LIN {X 0,Y 655.991,Z 1140.634,A -85,B 0,C 180,E1 30861.232,E2 30861.232} C_VEL
LIN {X 0,Y 656.124,Z 1133.603,A -85,B 0,C 180,E1 30859.285,E2 30859.285} C_VEL
LIN {X 0,Y 656.323,Z 1125.528,A -85,B 0,C 180,E1 30857.417,E2 30857.417} C_VEL
LIN {X 0,Y 656.666,Z 1114.351,A -85,B 0,C 180,E1 30855.269,E2 30855.269} C_VEL
LIN {X 0,Y 657.071,Z 1103.391,A -85,B 0,C 180,E1 30853.467,E2 30853.467} C_VEL
LIN {X 0,Y 657.695,Z 1089.324,A -85,B 0,C 180,E1 30851.473,E2 30851.473} C_VEL
LIN {X 0,Y 658.406,Z 1075.305,A -85,B 0,C 180,E1 30849.742,E2 30849.742} C_VEL
LIN {X 0,Y 659.336,Z 1058.307,A -85,B 0,C 180,E1 30847.908,E2 30847.908} C_VEL
LIN {X 0,Y 660.248,Z 1042.797,A -85,B 0,C 180,E1 30846.434,E2 30846.434} C_VEL
LIN {X 0,Y 661.459,Z 1022.865,A -85,B 0,C 180,E1 30844.768,E2 30844.768} C_VEL
LIN {X 0,Y 662.618,Z 1004.407,A -85,B 0,C 180,E1 30843.423,E2 30843.423} C_VEL
LIN {X 0,Y 663.968,Z 982.358,A -85,B 0,C 180,E1 30842.024,E2 30842.024} C_VEL
LIN {X 0,Y 665.114,Z 962.745,A -85,B 0,C 180,E1 30840.949,E2 30840.949} C_VEL
LIN {X 0,Y 666.461,Z 938.728,A -85,B 0,C 180,E1 30839.828,E2 30839.828} C_VEL
LIN {X 0,Y 667.412,Z 919.676,A -85,B 0,C 180,E1 30839.078,E2 30839.078} C_VEL
LIN {X 0,Y 668.429,Z 897.141,A -85,B 0,C 180,E1 30838.328,E2 30838.328} C_VEL
LIN {X 0,Y 669.288,Z 873.179,A -85,B 0,C 180,E1 30837.708,E2 30837.708} C_VEL
LIN {X 0,Y 670.004,Z 850.868,A -85,B 0,C 180,E1 30837.268,E2 30837.268} C_VEL
LIN {X 0,Y 670.501,Z 818.389,A -85,B 0,C 180,E1 30836.831,E2 30836.831} C_VEL
LIN {X 0,Y 672.565,Z 585.869,A -85,B 0,C 180,E1 30834.073,E2 30834.073} C_VEL
LIN {X 0,Y 673.662,Z 473.958,A -85,B 0,C 180,E1 30832.7,E2 30832.7} C_VEL
LIN {X 0,Y 669.198,Z 453.811,A -85,B 0,C 180,E1 30832.148,E2 30832.148} C_VEL
LIN {X 0,Y 669.234,Z 447.014,A -85,B 0,C 180,E1 30831.665,E2 30831.665} C_VEL
LIN {X 0,Y 660.986,Z 426.127,A -85,B 0,C 180,E1 30829.537,E2 30829.537} C_VEL
LIN {X 0,Y 656.734,Z 415.633,A -85,B 0,C 180,E1 30828.38,E2 30828.38} C_VEL
LIN {X 0,Y 656.685,Z 415.429,A -85,B 0,C 180,E1 30825.417,E2 30825.417} C_VEL
LIN {X 0,Y 656.705,Z 415.423,A -85,B 0,C 180,E1 30822.27,E2 30822.27} C_VEL
LIN {X 0,Y 656.674,Z 415.401,A -85,B 0,C 180,E1 30819.304,E2 30819.304} C_VEL
LIN {X 0,Y 656.707,Z 415.43,A -85,B 0,C 180,E1 30816.199,E2 30816.199} C_VEL
LIN {X 0,Y 656.676,Z 415.41,A -85,B 0,C 180,E1 30813.127,E2 30813.127} C_VEL
LIN {X 0,Y 656.705,Z 415.426,A -85,B 0,C 180,E1 30809.961,E2 30809.961} C_VEL
LIN {X 0,Y 656.674,Z 415.427,A -85,B 0,C 180,E1 30806.985,E2 30806.985} C_VEL
LIN {X 0,Y 656.691,Z 415.431,A -85,B 0,C 180,E1 30803.797,E2 30803.797} C_VEL
LIN {X 0,Y 656.667,Z 415.426,A -85,B 0,C 180,E1 30800.874,E2 30800.874} C_VEL
LIN {X 0,Y 656.69,Z 415.425,A -85,B 0,C 180,E1 30797.73,E2 30797.73} C_VEL
LIN {X 0,Y 656.658,Z 415.423,A -85,B 0,C 180,E1 30794.822,E2 30794.822} C_VEL
LIN {X 0,Y 656.692,Z 415.431,A -85,B 0,C 180,E1 30791.684,E2 30791.684} C_VEL
LIN {X 0,Y 656.651,Z 415.427,A -85,B 0,C 180,E1 30788.794,E2 30788.794} C_VEL
LIN {X 0,Y 656.706,Z 415.422,A -85,B 0,C 180,E1 30785.767,E2 30785.767} C_VEL
LIN {X 0,Y 656.64,Z 415.431,A -85,B 0,C 180,E1 30782.88,E2 30782.88} C_VEL
LIN {X 0,Y 656.715,Z 415.418,A -85,B 0,C 180,E1 30779.913,E2 30779.913} C_VEL
LIN {X 0,Y 656.637,Z 415.424,A -85,B 0,C 180,E1 30776.945,E2 30776.945} C_VEL
LIN {X 0,Y 656.657,Z 415.429,A -85,B 0,C 180,E1 30774.232,E2 30774.232} C_VEL
LIN {X 0,Y 656.644,Z 415.432,A -85,B 0,C 180,E1 30771.065,E2 30771.065} C_VEL
LIN {X 0,Y 656.632,Z 415.429,A -85,B 0,C 180,E1 30768.404,E2 30768.404} C_VEL
LIN {X 0,Y 656.685,Z 415.434,A -85,B 0,C 180,E1 30765.359,E2 30765.359} C_VEL
LIN {X 0,Y 656.619,Z 415.429,A -85,B 0,C 180,E1 30762.543,E2 30762.543} C_VEL
LIN {X 0,Y 656.677,Z 415.429,A -85,B 0,C 180,E1 30759.711,E2 30759.711} C_VEL
LIN {X 0,Y 656.619,Z 415.433,A -85,B 0,C 180,E1 30756.671,E2 30756.671} C_VEL
LIN {X 0,Y 656.619,Z 415.433,A -85,B 0,C 180,E1 30754.085,E2 30754.085} C_VEL
LIN {X 0,Y 656.657,Z 415.435,A -85,B 0,C 180,E1 30751.039,E2 30751.039} C_VEL
LIN {X 0,Y 656.603,Z 415.43,A -85,B 0,C 180,E1 30748.349,E2 30748.349} C_VEL
LIN {X 0,Y 656.63,Z 415.433,A -85,B 0,C 180,E1 30745.707,E2 30745.707} C_VEL
LIN {X 0,Y 656.621,Z 415.429,A -85,B 0,C 180,E1 30742.584,E2 30742.584} C_VEL
LIN {X 0,Y 656.627,Z 415.432,A -85,B 0,C 180,E1 30740.609,E2 30740.609} C_VEL
LIN {X 0,Y 655.592,Z 415.557,A -85,B 0,C 180,E1 30739.937,E2 30739.937} C_VEL
LIN {X 0,Y 649.186,Z 416.345,A -85,B 0,C 180,E1 30738.053,E2 30738.053} C_VEL
LIN {X 0,Y 648.701,Z 416.411,A -85,B 0,C 180,E1 30737.563,E2 30737.563} C_VEL
LIN {X 0,Y 648.688,Z 416.395,A -85,B 0,C 180,E1 30734.411,E2 30734.411} C_VEL
LIN {X 0,Y 648.685,Z 416.41,A -85,B 0,C 180,E1 30731.751,E2 30731.751} C_VEL
LIN {X 0,Y 648.793,Z 416.828,A -85,B 0,C 180,E1 30731.291,E2 30731.291} C_VEL
LIN {X 0,Y 657.127,Z 438.059,A -85,B 0,C 180,E1 30728.894,E2 30728.894} C_VEL
LIN {X 0,Y 661.622,Z 449.959,A -85,B 0,C 180,E1 30727.63,E2 30727.63} C_VEL
LIN {X 0,Y 659.646,Z 489.454,A -85,B 0,C 180,E1 30724.693,E2 30724.693} C_VEL
LIN {X 0,Y 659.389,Z 497.949,A -85,B 0,C 180,E1 30724.101,E2 30724.101} C_VEL
LIN {X 0,Y 664.297,Z 521.472,A -85,B 0,C 180,E1 30723.492,E2 30723.492} C_VEL
LIN {X 0,Y 661.38,Z 776.493,A -85,B 0,C 180,E1 30720.424,E2 30720.424} C_VEL
LIN {X 0,Y 660.462,Z 847.868,A -85,B 0,C 180,E1 30719.543,E2 30719.543} C_VEL
LIN {X 0,Y 659.772,Z 870.792,A -85,B 0,C 180,E1 30719.103,E2 30719.103} C_VEL
LIN {X 0,Y 658.928,Z 893.234,A -85,B 0,C 180,E1 30718.525,E2 30718.525} C_VEL
LIN {X 0,Y 657.886,Z 915.745,A -85,B 0,C 180,E1 30717.764,E2 30717.764} C_VEL
LIN {X 0,Y 656.714,Z 938.163,A -85,B 0,C 180,E1 30716.845,E2 30716.845} C_VEL
LIN {X 0,Y 655.667,Z 957.982,A -85,B 0,C 180,E1 30715.874,E2 30715.874} C_VEL
LIN {X 0,Y 654.496,Z 978.096,A -85,B 0,C 180,E1 30714.716,E2 30714.716} C_VEL
LIN {X 0,Y 653.41,Z 996.456,A -85,B 0,C 180,E1 30713.493,E2 30713.493} C_VEL
LIN {X 0,Y 652.29,Z 1014.965,A -85,B 0,C 180,E1 30712.059,E2 30712.059} C_VEL
LIN {X 0,Y 651.303,Z 1032.191,A -85,B 0,C 180,E1 30710.53,E2 30710.53} C_VEL
LIN {X 0,Y 650.415,Z 1047.757,A -85,B 0,C 180,E1 30708.928,E2 30708.928} C_VEL
LIN {X 0,Y 649.633,Z 1063.216,A -85,B 0,C 180,E1 30707.094,E2 30707.094} C_VEL
LIN {X 0,Y 649.074,Z 1075.943,A -85,B 0,C 180,E1 30705.345,E2 30705.345} C_VEL
LIN {X 0,Y 648.61,Z 1087.596,A -85,B 0,C 180,E1 30703.461,E2 30703.461} C_VEL
LIN {X 0,Y 648.305,Z 1097.6,A -85,B 0,C 180,E1 30701.566,E2 30701.566} C_VEL
LIN {X 0,Y 648.095,Z 1105.866,A -85,B 0,C 180,E1 30699.645,E2 30699.645} C_VEL
LIN {X 0,Y 647.972,Z 1112.927,A -85,B 0,C 180,E1 30697.626,E2 30697.626} C_VEL
LIN {X 0,Y 647.918,Z 1117.861,A -85,B 0,C 180,E1 30695.757,E2 30695.757} C_VEL
LIN {X 0,Y 647.899,Z 1121.718,A -85,B 0,C 180,E1 30693.716,E2 30693.716} C_VEL
LIN {X 0,Y 647.9,Z 1123.791,A -85,B 0,C 180,E1 30691.769,E2 30691.769} C_VEL
LIN {X 0,Y 647.896,Z 1124.426,A -85,B 0,C 180,E1 30689.646,E2 30689.646} C_VEL
LIN {X 0,Y 647.904,Z 1123.522,A -85,B 0,C 180,E1 30687.789,E2 30687.789} C_VEL
LIN {X 0,Y 647.909,Z 1120.86,A -85,B 0,C 180,E1 30685.663,E2 30685.663} C_VEL
LIN {X 0,Y 647.945,Z 1117.036,A -85,B 0,C 180,E1 30683.799,E2 30683.799} C_VEL
LIN {X 0,Y 648.021,Z 1110.906,A -85,B 0,C 180,E1 30681.66,E2 30681.66} C_VEL
LIN {X 0,Y 648.137,Z 1103.956,A -85,B 0,C 180,E1 30679.781,E2 30679.781} C_VEL
LIN {X 0,Y 648.371,Z 1094.872,A -85,B 0,C 180,E1 30677.803,E2 30677.803} C_VEL
LIN {X 0,Y 648.727,Z 1084.488,A -85,B 0,C 180,E1 30675.905,E2 30675.905} C_VEL
LIN {X 0,Y 649.19,Z 1072.616,A -85,B 0,C 180,E1 30674.088,E2 30674.088} C_VEL
LIN {X 0,Y 649.858,Z 1058.761,A -85,B 0,C 180,E1 30672.254,E2 30672.254} C_VEL
LIN {X 0,Y 650.604,Z 1044.342,A -85,B 0,C 180,E1 30670.612,E2 30670.612} C_VEL
LIN {X 0,Y 651.564,Z 1027.154,A -85,B 0,C 180,E1 30668.914,E2 30668.914} C_VEL
LIN {X 0,Y 652.618,Z 1009.902,A -85,B 0,C 180,E1 30667.431,E2 30667.431} C_VEL
LIN {X 0,Y 653.681,Z 991.704,A -85,B 0,C 180,E1 30666.087,E2 30666.087} C_VEL
LIN {X 0,Y 654.878,Z 971.864,A -85,B 0,C 180,E1 30664.812,E2 30664.812} C_VEL
LIN {X 0,Y 655.999,Z 951.829,A -85,B 0,C 180,E1 30663.718,E2 30663.718} C_VEL
LIN {X 0,Y 657.164,Z 929.599,A -85,B 0,C 180,E1 30662.695,E2 30662.695} C_VEL
LIN {X 0,Y 658.36,Z 905.845,A -85,B 0,C 180,E1 30661.789,E2 30661.789} C_VEL
LIN {X 0,Y 659.26,Z 884.849,A -85,B 0,C 180,E1 30661.154,E2 30661.154} C_VEL
LIN {X 0,Y 660.066,Z 862.091,A -85,B 0,C 180,E1 30660.619,E2 30660.619} C_VEL
LIN {X 0,Y 660.588,Z 840.006,A -85,B 0,C 180,E1 30660.256,E2 30660.256} C_VEL
LIN {X 0,Y 663.263,Z 610.425,A -85,B 0,C 180,E1 30657.486,E2 30657.486} C_VEL
LIN {X 0,Y 664.119,Z 519.815,A -85,B 0,C 180,E1 30656.386,E2 30656.386} C_VEL
LIN {X 0,Y 659.292,Z 497.129,A -85,B 0,C 180,E1 30655.773,E2 30655.773} C_VEL
LIN {X 0,Y 661.327,Z 455.954,A -85,B 0,C 180,E1 30652.732,E2 30652.732} C_VEL
LIN {X 0,Y 661.489,Z 449.538,A -85,B 0,C 180,E1 30652.238,E2 30652.238} C_VEL
LIN {X 0,Y 653.831,Z 429.55,A -85,B 0,C 180,E1 30650.08,E2 30650.08} C_VEL
LIN {X 0,Y 648.749,Z 416.581,A -85,B 0,C 180,E1 30648.569,E2 30648.569} C_VEL
LIN {X 0,Y 648.685,Z 416.396,A -85,B 0,C 180,E1 30645.788,E2 30645.788} C_VEL
LIN {X 0,Y 648.762,Z 416.412,A -85,B 0,C 180,E1 30642.808,E2 30642.808} C_VEL
LIN {X 0,Y 648.677,Z 416.419,A -85,B 0,C 180,E1 30639.884,E2 30639.884} C_VEL
LIN {X 0,Y 648.697,Z 416.411,A -85,B 0,C 180,E1 30637.284,E2 30637.284} C_VEL
LIN {X 0,Y 648.689,Z 416.424,A -85,B 0,C 180,E1 30634.13,E2 30634.13} C_VEL
LIN {X 0,Y 648.671,Z 416.419,A -85,B 0,C 180,E1 30631.504,E2 30631.504} C_VEL
LIN {X 0,Y 648.745,Z 416.415,A -85,B 0,C 180,E1 30628.535,E2 30628.535} C_VEL
LIN {X 0,Y 648.664,Z 416.424,A -85,B 0,C 180,E1 30625.61,E2 30625.61} C_VEL
LIN {X 0,Y 648.719,Z 416.423,A -85,B 0,C 180,E1 30622.821,E2 30622.821} C_VEL
LIN {X 0,Y 648.683,Z 416.422,A -85,B 0,C 180,E1 30619.823,E2 30619.823} C_VEL
LIN {X 0,Y 648.679,Z 416.419,A -85,B 0,C 180,E1 30617.215,E2 30617.215} C_VEL
LIN {X 0,Y 648.742,Z 416.418,A -85,B 0,C 180,E1 30614.186,E2 30614.186} C_VEL
LIN {X 0,Y 648.682,Z 416.42,A -85,B 0,C 180,E1 30611.378,E2 30611.378} C_VEL
LIN {X 0,Y 648.746,Z 416.412,A -85,B 0,C 180,E1 30608.509,E2 30608.509} C_VEL
LIN {X 0,Y 648.695,Z 416.42,A -85,B 0,C 180,E1 30605.484,E2 30605.484} C_VEL
LIN {X 0,Y 648.713,Z 416.413,A -85,B 0,C 180,E1 30602.739,E2 30602.739} C_VEL
LIN {X 0,Y 648.711,Z 416.409,A -85,B 0,C 180,E1 30599.558,E2 30599.558} C_VEL
LIN {X 0,Y 648.707,Z 416.422,A -85,B 0,C 180,E1 30596.819,E2 30596.819} C_VEL
LIN {X 0,Y 648.749,Z 416.415,A -85,B 0,C 180,E1 30593.718,E2 30593.718} C_VEL
LIN {X 0,Y 648.707,Z 416.418,A -85,B 0,C 180,E1 30590.865,E2 30590.865} C_VEL
LIN {X 0,Y 648.772,Z 416.415,A -85,B 0,C 180,E1 30587.81,E2 30587.81} C_VEL
LIN {X 0,Y 648.711,Z 416.414,A -85,B 0,C 180,E1 30584.901,E2 30584.901} C_VEL
LIN {X 0,Y 648.77,Z 416.408,A -85,B 0,C 180,E1 30581.954,E2 30581.954} C_VEL
LIN {X 0,Y 648.721,Z 416.416,A -85,B 0,C 180,E1 30578.953,E2 30578.953} C_VEL
LIN {X 0,Y 648.77,Z 416.421,A -85,B 0,C 180,E1 30575.991,E2 30575.991} C_VEL
LIN {X 0,Y 648.727,Z 416.417,A -85,B 0,C 180,E1 30572.856,E2 30572.856} C_VEL
LIN {X 0,Y 648.773,Z 416.414,A -85,B 0,C 180,E1 30569.941,E2 30569.941} C_VEL
LIN {X 0,Y 648.733,Z 416.396,A -85,B 0,C 180,E1 30566.817,E2 30566.817} C_VEL
LIN {X 0,Y 648.766,Z 416.418,A -85,B 0,C 180,E1 30563.822,E2 30563.822} C_VEL
LIN {X 0,Y 648.732,Z 416.388,A -85,B 0,C 180,E1 30560.691,E2 30560.691} C_VEL
LIN {X 0,Y 648.765,Z 416.41,A -85,B 0,C 180,E1 30557.661,E2 30557.661} C_VEL
LIN {X 0,Y 648.744,Z 416.419,A -85,B 0,C 180,E1 30554.53,E2 30554.53} C_VEL
LIN {X 0,Y 648.775,Z 416.622,A -85,B 0,C 180,E1 30552.156,E2 30552.156} C_VEL
LIN {X 0,Y 657.494,Z 438.049,A -85,B 0,C 180,E1 30549.81,E2 30549.81} C_VEL
LIN {X 0,Y 662.5,Z 451.205,A -85,B 0,C 180,E1 30548.477,E2 30548.477} C_VEL
LIN {X 0,Y 662.507,Z 454.848,A -85,B 0,C 180,E1 30548.253,E2 30548.253} C_VEL
LIN {X 0,Y 667.304,Z 477.152,A -85,B 0,C 180,E1 30547.654,E2 30547.654} C_VEL
LIN {X 0,Y 664.523,Z 721.617,A -85,B 0,C 180,E1 30544.669,E2 30544.669} C_VEL
LIN {X 0,Y 663.232,Z 844.483,A -85,B 0,C 180,E1 30543.181,E2 30543.181} C_VEL
LIN {X 0,Y 662.513,Z 870.087,A -85,B 0,C 180,E1 30542.714,E2 30542.714} C_VEL
LIN {X 0,Y 661.751,Z 891.398,A -85,B 0,C 180,E1 30542.194,E2 30542.194} C_VEL
LIN {X 0,Y 660.735,Z 914.535,A -85,B 0,C 180,E1 30541.473,E2 30541.473} C_VEL
LIN {X 0,Y 659.605,Z 935.33,A -85,B 0,C 180,E1 30540.671,E2 30540.671} C_VEL
LIN {X 0,Y 658.38,Z 957.268,A -85,B 0,C 180,E1 30539.677,E2 30539.677} C_VEL
LIN {X 0,Y 656.936,Z 979.114,A -85,B 0,C 180,E1 30538.5,E2 30538.5} C_VEL
LIN {X 0,Y 655.616,Z 999.646,A -85,B 0,C 180,E1 30537.228,E2 30537.228} C_VEL
LIN {X 0,Y 654.268,Z 1019.215,A -85,B 0,C 180,E1 30535.821,E2 30535.821} C_VEL
LIN {X 0,Y 653.067,Z 1037.201,A -85,B 0,C 180,E1 30534.357,E2 30534.357} C_VEL
LIN {X 0,Y 651.924,Z 1054.602,A -85,B 0,C 180,E1 30532.737,E2 30532.737} C_VEL
LIN {X 0,Y 650.985,Z 1069.628,A -85,B 0,C 180,E1 30531.159,E2 30531.159} C_VEL
LIN {X 0,Y 650.057,Z 1086.032,A -85,B 0,C 180,E1 30529.19,E2 30529.19} C_VEL
LIN {X 0,Y 649.404,Z 1099.154,A -85,B 0,C 180,E1 30527.38,E2 30527.38} C_VEL
LIN {X 0,Y 648.819,Z 1112.382,A -85,B 0,C 180,E1 30525.263,E2 30525.263} C_VEL
LIN {X 0,Y 648.448,Z 1122.48,A -85,B 0,C 180,E1 30523.373,E2 30523.373} C_VEL
LIN {X 0,Y 648.165,Z 1132.189,A -85,B 0,C 180,E1 30521.208,E2 30521.208} C_VEL
LIN {X 0,Y 648.053,Z 1138.817,A -85,B 0,C 180,E1 30519.413,E2 30519.413} C_VEL
LIN {X 0,Y 647.946,Z 1145.243,A -85,B 0,C 180,E1 30517.27,E2 30517.27} C_VEL
LIN {X 0,Y 647.896,Z 1149.656,A -85,B 0,C 180,E1 30515.224,E2 30515.224} C_VEL
LIN {X 0,Y 647.904,Z 1152.463,A -85,B 0,C 180,E1 30513.362,E2 30513.362} C_VEL
LIN {X 0,Y 647.909,Z 1154.215,A -85,B 0,C 180,E1 30511.15,E2 30511.15} C_VEL
LIN {X 0,Y 647.885,Z 1154.328,A -85,B 0,C 180,E1 30509.293,E2 30509.293} C_VEL
LIN {X 0,Y 647.888,Z 1153.225,A -85,B 0,C 180,E1 30507.346,E2 30507.346} C_VEL
LIN {X 0,Y 647.903,Z 1150.292,A -85,B 0,C 180,E1 30505.131,E2 30505.131} C_VEL
LIN {X 0,Y 647.939,Z 1146.689,A -85,B 0,C 180,E1 30503.354,E2 30503.354} C_VEL
LIN {X 0,Y 648,Z 1140.935,A -85,B 0,C 180,E1 30501.213,E2 30501.213} C_VEL
LIN {X 0,Y 648.142,Z 1133.603,A -85,B 0,C 180,E1 30499.152,E2 30499.152} C_VEL
LIN {X 0,Y 648.372,Z 1125.529,A -85,B 0,C 180,E1 30497.26,E2 30497.26} C_VEL
LIN {X 0,Y 648.748,Z 1114.436,A -85,B 0,C 180,E1 30495.1,E2 30495.1} C_VEL
LIN {X 0,Y 649.198,Z 1103.393,A -85,B 0,C 180,E1 30493.261,E2 30493.261} C_VEL
LIN {X 0,Y 649.877,Z 1089.323,A -85,B 0,C 180,E1 30491.242,E2 30491.242} C_VEL
LIN {X 0,Y 650.67,Z 1075.307,A -85,B 0,C 180,E1 30489.49,E2 30489.49} C_VEL
LIN {X 0,Y 651.686,Z 1058.305,A -85,B 0,C 180,E1 30487.635,E2 30487.635} C_VEL
LIN {X 0,Y 652.726,Z 1042.29,A -85,B 0,C 180,E1 30486.098,E2 30486.098} C_VEL
LIN {X 0,Y 654.04,Z 1022.359,A -85,B 0,C 180,E1 30484.421,E2 30484.421} C_VEL
LIN {X 0,Y 655.275,Z 1004.392,A -85,B 0,C 180,E1 30483.1,E2 30483.1} C_VEL
LIN {X 0,Y 656.73,Z 982.354,A -85,B 0,C 180,E1 30481.688,E2 30481.688} C_VEL
LIN {X 0,Y 657.988,Z 962.741,A -85,B 0,C 180,E1 30480.604,E2 30480.604} C_VEL
LIN {X 0,Y 659.437,Z 938.724,A -85,B 0,C 180,E1 30479.472,E2 30479.472} C_VEL
LIN {X 0,Y 660.468,Z 919.672,A -85,B 0,C 180,E1 30478.716,E2 30478.716} C_VEL
LIN {X 0,Y 661.503,Z 898.098,A -85,B 0,C 180,E1 30477.993,E2 30477.993} C_VEL
LIN {X 0,Y 662.367,Z 873.835,A -85,B 0,C 180,E1 30477.367,E2 30477.367} C_VEL
LIN {X 0,Y 663.055,Z 851.771,A -85,B 0,C 180,E1 30476.935,E2 30476.935} C_VEL
LIN {X 0,Y 663.553,Z 819.351,A -85,B 0,C 180,E1 30476.498,E2 30476.498} C_VEL
LIN {X 0,Y 665.842,Z 590.197,A -85,B 0,C 180,E1 30473.746,E2 30473.746} C_VEL
LIN {X 0,Y 667.088,Z 475.51,A -85,B 0,C 180,E1 30472.318,E2 30472.318} C_VEL
LIN {X 0,Y 662.402,Z 454.038,A -85,B 0,C 180,E1 30471.715,E2 30471.715} C_VEL
LIN {X 0,Y 662.299,Z 450.377,A -85,B 0,C 180,E1 30471.448,E2 30471.448} C_VEL
LIN {X 0,Y 654.091,Z 429.742,A -85,B 0,C 180,E1 30469.308,E2 30469.308} C_VEL
LIN {X 0,Y 648.773,Z 416.612,A -85,B 0,C 180,E1 30467.839,E2 30467.839} C_VEL
LIN {X 0,Y 648.763,Z 416.396,A -85,B 0,C 180,E1 30464.777,E2 30464.777} C_VEL
LIN {X 0,Y 648.743,Z 416.422,A -85,B 0,C 180,E1 30461.746,E2 30461.746} C_VEL
LIN {X 0,Y 648.767,Z 416.388,A -85,B 0,C 180,E1 30458.736,E2 30458.736} C_VEL
LIN {X 0,Y 648.736,Z 416.411,A -85,B 0,C 180,E1 30455.634,E2 30455.634} C_VEL
LIN {X 0,Y 648.767,Z 416.398,A -85,B 0,C 180,E1 30452.54,E2 30452.54} C_VEL
LIN {X 0,Y 648.733,Z 416.412,A -85,B 0,C 180,E1 30449.552,E2 30449.552} C_VEL
LIN {X 0,Y 648.768,Z 416.414,A -85,B 0,C 180,E1 30446.548,E2 30446.548} C_VEL
LIN {X 0,Y 648.725,Z 416.417,A -85,B 0,C 180,E1 30443.432,E2 30443.432} C_VEL
LIN {X 0,Y 648.767,Z 416.413,A -85,B 0,C 180,E1 30440.436,E2 30440.436} C_VEL
LIN {X 0,Y 648.721,Z 416.419,A -85,B 0,C 180,E1 30437.306,E2 30437.306} C_VEL
LIN {X 0,Y 648.763,Z 416.409,A -85,B 0,C 180,E1 30434.367,E2 30434.367} C_VEL
LIN {X 0,Y 648.718,Z 416.417,A -85,B 0,C 180,E1 30431.289,E2 30431.289} C_VEL
LIN {X 0,Y 648.738,Z 416.414,A -85,B 0,C 180,E1 30428.42,E2 30428.42} C_VEL
LIN {X 0,Y 648.719,Z 416.414,A -85,B 0,C 180,E1 30425.306,E2 30425.306} C_VEL
LIN {X 0,Y 648.719,Z 416.418,A -85,B 0,C 180,E1 30422.474,E2 30422.474} C_VEL
LIN {X 0,Y 648.714,Z 416.422,A -85,B 0,C 180,E1 30419.205,E2 30419.205} C_VEL
LIN {X 0,Y 648.704,Z 416.41,A -85,B 0,C 180,E1 30416.465,E2 30416.465} C_VEL
LIN {X 0,Y 648.735,Z 416.418,A -85,B 0,C 180,E1 30413.362,E2 30413.362} C_VEL
LIN {X 0,Y 648.69,Z 416.419,A -85,B 0,C 180,E1 30410.575,E2 30410.575} C_VEL
LIN {X 0,Y 648.768,Z 416.41,A -85,B 0,C 180,E1 30407.63,E2 30407.63} C_VEL
LIN {X 0,Y 648.685,Z 416.422,A -85,B 0,C 180,E1 30404.717,E2 30404.717} C_VEL
LIN {X 0,Y 648.703,Z 416.417,A -85,B 0,C 180,E1 30402.045,E2 30402.045} C_VEL
LIN {X 0,Y 648.69,Z 416.42,A -85,B 0,C 180,E1 30398.836,E2 30398.836} C_VEL
LIN {X 0,Y 648.676,Z 416.422,A -85,B 0,C 180,E1 30396.277,E2 30396.277} C_VEL
LIN {X 0,Y 648.758,Z 416.422,A -85,B 0,C 180,E1 30393.352,E2 30393.352} C_VEL
LIN {X 0,Y 648.668,Z 416.426,A -85,B 0,C 180,E1 30390.444,E2 30390.444} C_VEL
LIN {X 0,Y 648.679,Z 416.419,A -85,B 0,C 180,E1 30387.873,E2 30387.873} C_VEL
LIN {X 0,Y 648.677,Z 416.397,A -85,B 0,C 180,E1 30384.629,E2 30384.629} C_VEL
LIN {X 0,Y 648.671,Z 416.423,A -85,B 0,C 180,E1 30381.969,E2 30381.969} C_VEL
LIN {X 0,Y 648.75,Z 416.39,A -85,B 0,C 180,E1 30379.045,E2 30379.045} C_VEL
LIN {X 0,Y 648.701,Z 416.411,A -85,B 0,C 180,E1 30377.563,E2 30377.563} C_VEL
LIN {X 0,Y 647.769,Z 416.544,A -85,B 0,C 180,E1 30376.882,E2 30376.882} C_VEL
LIN {X 0,Y 641.223,Z 417.33,A -85,B 0,C 180,E1 30374.926,E2 30374.926} C_VEL
LIN {X 0,Y 640.754,Z 417.382,A -85,B 0,C 180,E1 30374.479,E2 30374.479} C_VEL
LIN {X 0,Y 640.771,Z 417.624,A -85,B 0,C 180,E1 30371.884,E2 30371.884} C_VEL
LIN {X 0,Y 647.744,Z 434.924,A -85,B 0,C 180,E1 30369.838,E2 30369.838} C_VEL
LIN {X 0,Y 654.667,Z 453.446,A -85,B 0,C 180,E1 30367.829,E2 30367.829} C_VEL
LIN {X 0,Y 652.477,Z 493.787,A -85,B 0,C 180,E1 30364.804,E2 30364.804} C_VEL
LIN {X 0,Y 652.502,Z 497.976,A -85,B 0,C 180,E1 30364.541,E2 30364.541} C_VEL
LIN {X 0,Y 657.764,Z 522.777,A -85,B 0,C 180,E1 30363.881,E2 30363.881} C_VEL
LIN {X 0,Y 654.701,Z 777.349,A -85,B 0,C 180,E1 30360.801,E2 30360.801} C_VEL
LIN {X 0,Y 653.739,Z 847.737,A -85,B 0,C 180,E1 30359.926,E2 30359.926} C_VEL
LIN {X 0,Y 653.008,Z 870.705,A -85,B 0,C 180,E1 30359.485,E2 30359.485} C_VEL
LIN {X 0,Y 652.101,Z 893.018,A -85,B 0,C 180,E1 30358.908,E2 30358.908} C_VEL
LIN {X 0,Y 651.019,Z 914.402,A -85,B 0,C 180,E1 30358.183,E2 30358.183} C_VEL
LIN {X 0,Y 649.85,Z 935.051,A -85,B 0,C 180,E1 30357.341,E2 30357.341} C_VEL
LIN {X 0,Y 648.508,Z 955.763,A -85,B 0,C 180,E1 30356.313,E2 30356.313} C_VEL
LIN {X 0,Y 647.181,Z 976.91,A -85,B 0,C 180,E1 30355.094,E2 30355.094} C_VEL
LIN {X 0,Y 645.987,Z 995.125,A -85,B 0,C 180,E1 30353.876,E2 30353.876} C_VEL
LIN {X 0,Y 644.782,Z 1013.861,A -85,B 0,C 180,E1 30352.426,E2 30352.426} C_VEL
LIN {X 0,Y 643.707,Z 1030.678,A -85,B 0,C 180,E1 30350.933,E2 30350.933} C_VEL
LIN {X 0,Y 642.762,Z 1046.071,A -85,B 0,C 180,E1 30349.351,E2 30349.351} C_VEL
LIN {X 0,Y 641.976,Z 1060.383,A -85,B 0,C 180,E1 30347.681,E2 30347.681} C_VEL
LIN {X 0,Y 641.29,Z 1073.264,A -85,B 0,C 180,E1 30345.927,E2 30345.927} C_VEL
LIN {X 0,Y 640.763,Z 1085.535,A -85,B 0,C 180,E1 30343.997,E2 30343.997} C_VEL
LIN {X 0,Y 640.407,Z 1095.334,A -85,B 0,C 180,E1 30342.168,E2 30342.168} C_VEL
LIN {X 0,Y 640.141,Z 1104.666,A -85,B 0,C 180,E1 30340.075,E2 30340.075} C_VEL
LIN {X 0,Y 640.017,Z 1111.514,A -85,B 0,C 180,E1 30338.173,E2 30338.173} C_VEL
LIN {X 0,Y 639.943,Z 1117.24,A -85,B 0,C 180,E1 30336.099,E2 30336.099} C_VEL
LIN {X 0,Y 639.913,Z 1121.019,A -85,B 0,C 180,E1 30334.212,E2 30334.212} C_VEL
LIN {X 0,Y 639.906,Z 1123.518,A -85,B 0,C 180,E1 30332.149,E2 30332.149} C_VEL
LIN {X 0,Y 639.903,Z 1124.448,A -85,B 0,C 180,E1 30330.179,E2 30330.179} C_VEL
LIN {X 0,Y 639.903,Z 1123.793,A -85,B 0,C 180,E1 30328.12,E2 30328.12} C_VEL
LIN {X 0,Y 639.905,Z 1121.72,A -85,B 0,C 180,E1 30326.147,E2 30326.147} C_VEL
LIN {X 0,Y 639.928,Z 1117.86,A -85,B 0,C 180,E1 30324.081,E2 30324.081} C_VEL
LIN {X 0,Y 639.986,Z 1112.673,A -85,B 0,C 180,E1 30322.097,E2 30322.097} C_VEL
LIN {X 0,Y 640.116,Z 1105.723,A -85,B 0,C 180,E1 30320.106,E2 30320.106} C_VEL
LIN {X 0,Y 640.344,Z 1097.595,A -85,B 0,C 180,E1 30318.196,E2 30318.196} C_VEL
LIN {X 0,Y 640.681,Z 1087.588,A -85,B 0,C 180,E1 30316.277,E2 30316.277} C_VEL
LIN {X 0,Y 641.17,Z 1076.426,A -85,B 0,C 180,E1 30314.441,E2 30314.441} C_VEL
LIN {X 0,Y 641.773,Z 1063.874,A -85,B 0,C 180,E1 30312.688,E2 30312.688} C_VEL
LIN {X 0,Y 642.572,Z 1049.415,A -85,B 0,C 180,E1 30310.927,E2 30310.927} C_VEL
LIN {X 0,Y 643.478,Z 1034.403,A -85,B 0,C 180,E1 30309.345,E2 30309.345} C_VEL
LIN {X 0,Y 644.603,Z 1016.532,A -85,B 0,C 180,E1 30307.709,E2 30307.709} C_VEL
LIN {X 0,Y 645.807,Z 998.347,A -85,B 0,C 180,E1 30306.262,E2 30306.262} C_VEL
LIN {X 0,Y 646.985,Z 979.741,A -85,B 0,C 180,E1 30304.996,E2 30304.996} C_VEL
LIN {X 0,Y 648.297,Z 959.455,A -85,B 0,C 180,E1 30303.794,E2 30303.794} C_VEL
LIN {X 0,Y 649.514,Z 939.785,A -85,B 0,C 180,E1 30302.792,E2 30302.792} C_VEL
LIN {X 0,Y 650.842,Z 917.92,A -85,B 0,C 180,E1 30301.859,E2 30301.859} C_VEL
LIN {X 0,Y 651.836,Z 898.37,A -85,B 0,C 180,E1 30301.174,E2 30301.174} C_VEL
LIN {X 0,Y 652.833,Z 875.117,A -85,B 0,C 180,E1 30300.526,E2 30300.526} C_VEL
LIN {X 0,Y 653.552,Z 853.926,A -85,B 0,C 180,E1 30300.088,E2 30300.088} C_VEL
LIN {X 0,Y 654.137,Z 823.568,A -85,B 0,C 180,E1 30299.667,E2 30299.667} C_VEL
LIN {X 0,Y 656.911,Z 591.86,A -85,B 0,C 180,E1 30296.864,E2 30296.864} C_VEL
LIN {X 0,Y 657.58,Z 521.351,A -85,B 0,C 180,E1 30295.999,E2 30295.999} C_VEL
LIN {X 0,Y 652.34,Z 496.691,A -85,B 0,C 180,E1 30295.316,E2 30295.316} C_VEL
LIN {X 0,Y 654.5,Z 456.495,A -85,B 0,C 180,E1 30292.313,E2 30292.313} C_VEL
LIN {X 0,Y 654.531,Z 452.855,A -85,B 0,C 180,E1 30292.024,E2 30292.024} C_VEL
LIN {X 0,Y 646.997,Z 433.261,A -85,B 0,C 180,E1 30289.876,E2 30289.876} C_VEL
LIN {X 0,Y 641.853,Z 420.538,A -85,B 0,C 180,E1 30288.396,E2 30288.396} C_VEL
LIN {X 0,Y 640.771,Z 417.564,A -85,B 0,C 180,E1 30288.006,E2 30288.006} C_VEL
LIN {X 0,Y 640.788,Z 417.379,A -85,B 0,C 180,E1 30285.234,E2 30285.234} C_VEL
LIN {X 0,Y 640.747,Z 417.395,A -85,B 0,C 180,E1 30282.146,E2 30282.146} C_VEL
LIN {X 0,Y 640.744,Z 417.408,A -85,B 0,C 180,E1 30279.546,E2 30279.546} C_VEL
LIN {X 0,Y 640.784,Z 417.377,A -85,B 0,C 180,E1 30276.479,E2 30276.479} C_VEL
LIN {X 0,Y 640.733,Z 417.413,A -85,B 0,C 180,E1 30273.642,E2 30273.642} C_VEL
LIN {X 0,Y 640.819,Z 417.404,A -85,B 0,C 180,E1 30270.679,E2 30270.679} C_VEL
LIN {X 0,Y 640.725,Z 417.41,A -85,B 0,C 180,E1 30267.713,E2 30267.713} C_VEL
LIN {X 0,Y 640.769,Z 417.408,A -85,B 0,C 180,E1 30264.918,E2 30264.918} C_VEL
LIN {X 0,Y 640.743,Z 417.409,A -85,B 0,C 180,E1 30261.899,E2 30261.899} C_VEL
LIN {X 0,Y 640.741,Z 417.412,A -85,B 0,C 180,E1 30259.225,E2 30259.225} C_VEL
LIN {X 0,Y 640.787,Z 417.407,A -85,B 0,C 180,E1 30256.126,E2 30256.126} C_VEL
LIN {X 0,Y 640.74,Z 417.408,A -85,B 0,C 180,E1 30253.354,E2 30253.354} C_VEL
LIN {X 0,Y 640.821,Z 417.411,A -85,B 0,C 180,E1 30250.428,E2 30250.428} C_VEL
LIN {X 0,Y 640.75,Z 417.404,A -85,B 0,C 180,E1 30247.442,E2 30247.442} C_VEL
LIN {X 0,Y 640.776,Z 417.411,A -85,B 0,C 180,E1 30244.744,E2 30244.744} C_VEL
LIN {X 0,Y 640.767,Z 417.409,A -85,B 0,C 180,E1 30241.52,E2 30241.52} C_VEL
LIN {X 0,Y 640.765,Z 417.399,A -85,B 0,C 180,E1 30238.838,E2 30238.838} C_VEL
LIN {X 0,Y 640.801,Z 417.4,A -85,B 0,C 180,E1 30235.705,E2 30235.705} C_VEL
LIN {X 0,Y 640.765,Z 417.408,A -85,B 0,C 180,E1 30232.919,E2 30232.919} C_VEL
LIN {X 0,Y 640.829,Z 417.398,A -85,B 0,C 180,E1 30229.845,E2 30229.845} C_VEL
LIN {X 0,Y 640.771,Z 417.407,A -85,B 0,C 180,E1 30226.923,E2 30226.923} C_VEL
LIN {X 0,Y 640.835,Z 417.407,A -85,B 0,C 180,E1 30223.968,E2 30223.968} C_VEL
LIN {X 0,Y 640.777,Z 417.402,A -85,B 0,C 180,E1 30220.871,E2 30220.871} C_VEL
LIN {X 0,Y 640.835,Z 417.397,A -85,B 0,C 180,E1 30217.912,E2 30217.912} C_VEL
LIN {X 0,Y 640.785,Z 417.404,A -85,B 0,C 180,E1 30214.829,E2 30214.829} C_VEL
LIN {X 0,Y 640.831,Z 417.402,A -85,B 0,C 180,E1 30211.785,E2 30211.785} C_VEL
LIN {X 0,Y 640.793,Z 417.408,A -85,B 0,C 180,E1 30208.771,E2 30208.771} C_VEL
LIN {X 0,Y 640.826,Z 417.373,A -85,B 0,C 180,E1 30205.717,E2 30205.717} C_VEL
LIN {X 0,Y 640.796,Z 417.409,A -85,B 0,C 180,E1 30202.628,E2 30202.628} C_VEL
LIN {X 0,Y 640.825,Z 417.383,A -85,B 0,C 180,E1 30199.644,E2 30199.644} C_VEL
LIN {X 0,Y 640.801,Z 417.381,A -85,B 0,C 180,E1 30196.641,E2 30196.641} C_VEL
LIN {X 0,Y 640.826,Z 417.395,A -85,B 0,C 180,E1 30193.603,E2 30193.603} C_VEL
LIN {X 0,Y 640.849,Z 417.645,A -85,B 0,C 180,E1 30192.702,E2 30192.702} C_VEL
LIN {X 0,Y 649.808,Z 439.556,A -85,B 0,C 180,E1 30190.251,E2 30190.251} C_VEL
LIN {X 0,Y 655.66,Z 454.735,A -85,B 0,C 180,E1 30188.701,E2 30188.701} C_VEL
LIN {X 0,Y 660.778,Z 478.855,A -85,B 0,C 180,E1 30188.038,E2 30188.038} C_VEL
LIN {X 0,Y 657.678,Z 724.431,A -85,B 0,C 180,E1 30185.001,E2 30185.001} C_VEL
LIN {X 0,Y 656.279,Z 844.479,A -85,B 0,C 180,E1 30183.529,E2 30183.529} C_VEL
LIN {X 0,Y 655.515,Z 869.939,A -85,B 0,C 180,E1 30183.059,E2 30183.059} C_VEL
LIN {X 0,Y 654.702,Z 891.147,A -85,B 0,C 180,E1 30182.537,E2 30182.537} C_VEL
LIN {X 0,Y 653.575,Z 916.157,A -85,B 0,C 180,E1 30181.755,E2 30181.755} C_VEL
LIN {X 0,Y 652.517,Z 936.172,A -85,B 0,C 180,E1 30180.989,E2 30180.989} C_VEL
LIN {X 0,Y 651.468,Z 954.258,A -85,B 0,C 180,E1 30180.176,E2 30180.176} C_VEL
LIN {X 0,Y 649.893,Z 977.307,A -85,B 0,C 180,E1 30178.95,E2 30178.95} C_VEL
LIN {X 0,Y 648.558,Z 995.776,A -85,B 0,C 180,E1 30177.813,E2 30177.813} C_VEL
LIN {X 0,Y 647.006,Z 1017.327,A -85,B 0,C 180,E1 30176.285,E2 30176.285} C_VEL
LIN {X 0,Y 645.76,Z 1034.285,A -85,B 0,C 180,E1 30174.908,E2 30174.908} C_VEL
LIN {X 0,Y 644.45,Z 1052.748,A -85,B 0,C 180,E1 30173.209,E2 30173.209} C_VEL
LIN {X 0,Y 643.41,Z 1067.936,A -85,B 0,C 180,E1 30171.612,E2 30171.612} C_VEL
LIN {X 0,Y 642.437,Z 1083.7,A -85,B 0,C 180,E1 30169.739,E2 30169.739} C_VEL
LIN {X 0,Y 641.633,Z 1097.247,A -85,B 0,C 180,E1 30167.878,E2 30167.878} C_VEL
LIN {X 0,Y 641.039,Z 1109.688,A -85,B 0,C 180,E1 30165.934,E2 30165.934} C_VEL
LIN {X 0,Y 640.574,Z 1120.643,A -85,B 0,C 180,E1 30163.909,E2 30163.909} C_VEL
LIN {X 0,Y 640.286,Z 1129.991,A -85,B 0,C 180,E1 30161.896,E2 30161.896} C_VEL
LIN {X 0,Y 640.071,Z 1137.907,A -85,B 0,C 180,E1 30159.804,E2 30159.804} C_VEL
LIN {X 0,Y 639.966,Z 1143.744,A -85,B 0,C 180,E1 30157.903,E2 30157.903} C_VEL
LIN {X 0,Y 639.919,Z 1149.016,A -85,B 0,C 180,E1 30155.649,E2 30155.649} C_VEL
LIN {X 0,Y 639.913,Z 1152.124,A -85,B 0,C 180,E1 30153.673,E2 30153.673} C_VEL
LIN {X 0,Y 639.898,Z 1154.102,A -85,B 0,C 180,E1 30151.522,E2 30151.522} C_VEL
LIN {X 0,Y 639.884,Z 1154.373,A -85,B 0,C 180,E1 30149.463,E2 30149.463} C_VEL
LIN {X 0,Y 639.903,Z 1153.429,A -85,B 0,C 180,E1 30147.582,E2 30147.582} C_VEL
LIN {X 0,Y 639.917,Z 1150.768,A -85,B 0,C 180,E1 30145.339,E2 30145.339} C_VEL
LIN {X 0,Y 639.941,Z 1146.896,A -85,B 0,C 180,E1 30143.36,E2 30143.36} C_VEL
LIN {X 0,Y 640.002,Z 1141.71,A -85,B 0,C 180,E1 30141.374,E2 30141.374} C_VEL
LIN {X 0,Y 640.156,Z 1134.309,A -85,B 0,C 180,E1 30139.197,E2 30139.197} C_VEL
LIN {X 0,Y 640.392,Z 1126.346,A -85,B 0,C 180,E1 30137.282,E2 30137.282} C_VEL
LIN {X 0,Y 640.799,Z 1115.377,A -85,B 0,C 180,E1 30135.08,E2 30135.08} C_VEL
LIN {X 0,Y 641.281,Z 1104.381,A -85,B 0,C 180,E1 30133.208,E2 30133.208} C_VEL
LIN {X 0,Y 642.037,Z 1090.021,A -85,B 0,C 180,E1 30131.099,E2 30131.099} C_VEL
LIN {X 0,Y 642.839,Z 1076.848,A -85,B 0,C 180,E1 30129.419,E2 30129.419} C_VEL
LIN {X 0,Y 643.936,Z 1060.155,A -85,B 0,C 180,E1 30127.543,E2 30127.543} C_VEL
LIN {X 0,Y 645.033,Z 1044.316,A -85,B 0,C 180,E1 30125.989,E2 30125.989} C_VEL
LIN {X 0,Y 646.36,Z 1026.198,A -85,B 0,C 180,E1 30124.406,E2 30124.406} C_VEL
LIN {X 0,Y 647.746,Z 1007.052,A -85,B 0,C 180,E1 30122.96,E2 30122.96} C_VEL
LIN {X 0,Y 649.227,Z 987.158,A -85,B 0,C 180,E1 30121.632,E2 30121.632} C_VEL
LIN {X 0,Y 650.633,Z 966.296,A -85,B 0,C 180,E1 30120.439,E2 30120.439} C_VEL
LIN {X 0,Y 651.976,Z 946.208,A -85,B 0,C 180,E1 30119.443,E2 30119.443} C_VEL
LIN {X 0,Y 653.244,Z 922.99,A -85,B 0,C 180,E1 30118.493,E2 30118.493} C_VEL
LIN {X 0,Y 654.23,Z 902.293,A -85,B 0,C 180,E1 30117.791,E2 30117.791} C_VEL
LIN {X 0,Y 655.202,Z 878.363,A -85,B 0,C 180,E1 30117.128,E2 30117.128} C_VEL
LIN {X 0,Y 655.961,Z 855.305,A -85,B 0,C 180,E1 30116.652,E2 30116.652} C_VEL
LIN {X 0,Y 656.528,Z 830.37,A -85,B 0,C 180,E1 30116.278,E2 30116.278} C_VEL
LIN {X 0,Y 659.107,Z 598.469,A -85,B 0,C 180,E1 30113.459,E2 30113.459} C_VEL
LIN {X 0,Y 660.573,Z 477.158,A -85,B 0,C 180,E1 30111.932,E2 30111.932} C_VEL
LIN {X 0,Y 655.599,Z 454.284,A -85,B 0,C 180,E1 30111.272,E2 30111.272} C_VEL
LIN {X 0,Y 647.214,Z 433.244,A -85,B 0,C 180,E1 30109.066,E2 30109.066} C_VEL
LIN {X 0,Y 641.513,Z 419.82,A -85,B 0,C 180,E1 30107.554,E2 30107.554} C_VEL
LIN {X 0,Y 640.833,Z 417.528,A -85,B 0,C 180,E1 30107.255,E2 30107.255} C_VEL
LIN {X 0,Y 640.814,Z 417.376,A -85,B 0,C 180,E1 30103.976,E2 30103.976} C_VEL
LIN {X 0,Y 640.833,Z 417.397,A -85,B 0,C 180,E1 30100.822,E2 30100.822} C_VEL
LIN {X 0,Y 640.801,Z 417.401,A -85,B 0,C 180,E1 30097.71,E2 30097.71} C_VEL
LIN {X 0,Y 640.826,Z 417.379,A -85,B 0,C 180,E1 30094.685,E2 30094.685} C_VEL
LIN {X 0,Y 640.796,Z 417.411,A -85,B 0,C 180,E1 30091.573,E2 30091.573} C_VEL
LIN {X 0,Y 640.834,Z 417.397,A -85,B 0,C 180,E1 30088.519,E2 30088.519} C_VEL
LIN {X 0,Y 640.788,Z 417.406,A -85,B 0,C 180,E1 30085.411,E2 30085.411} C_VEL
LIN {X 0,Y 640.834,Z 417.398,A -85,B 0,C 180,E1 30082.378,E2 30082.378} C_VEL
LIN {X 0,Y 640.783,Z 417.403,A -85,B 0,C 180,E1 30079.318,E2 30079.318} C_VEL
LIN {X 0,Y 640.83,Z 417.403,A -85,B 0,C 180,E1 30076.311,E2 30076.311} C_VEL
LIN {X 0,Y 640.778,Z 417.408,A -85,B 0,C 180,E1 30073.261,E2 30073.261} C_VEL
LIN {X 0,Y 640.815,Z 417.401,A -85,B 0,C 180,E1 30070.337,E2 30070.337} C_VEL
LIN {X 0,Y 640.778,Z 417.409,A -85,B 0,C 180,E1 30067.261,E2 30067.261} C_VEL
LIN {X 0,Y 640.783,Z 417.401,A -85,B 0,C 180,E1 30064.475,E2 30064.475} C_VEL
LIN {X 0,Y 640.777,Z 417.399,A -85,B 0,C 180,E1 30061.252,E2 30061.252} C_VEL
LIN {X 0,Y 640.765,Z 417.409,A -85,B 0,C 180,E1 30058.569,E2 30058.569} C_VEL
LIN {X 0,Y 640.802,Z 417.404,A -85,B 0,C 180,E1 30055.436,E2 30055.436} C_VEL
LIN {X 0,Y 640.753,Z 417.404,A -85,B 0,C 180,E1 30052.648,E2 30052.648} C_VEL
LIN {X 0,Y 640.83,Z 417.408,A -85,B 0,C 180,E1 30049.663,E2 30049.663} C_VEL
LIN {X 0,Y 640.748,Z 417.408,A -85,B 0,C 180,E1 30046.739,E2 30046.739} C_VEL
LIN {X 0,Y 640.761,Z 417.409,A -85,B 0,C 180,E1 30044.152,E2 30044.152} C_VEL
LIN {X 0,Y 640.754,Z 417.412,A -85,B 0,C 180,E1 30040.87,E2 30040.87} C_VEL
LIN {X 0,Y 640.744,Z 417.408,A -85,B 0,C 180,E1 30038.198,E2 30038.198} C_VEL
LIN {X 0,Y 640.794,Z 417.404,A -85,B 0,C 180,E1 30035.181,E2 30035.181} C_VEL
LIN {X 0,Y 640.732,Z 417.409,A -85,B 0,C 180,E1 30032.388,E2 30032.388} C_VEL
LIN {X 0,Y 640.774,Z 417.415,A -85,B 0,C 180,E1 30029.63,E2 30029.63} C_VEL
LIN {X 0,Y 640.734,Z 417.414,A -85,B 0,C 180,E1 30026.573,E2 30026.573} C_VEL
LIN {X 0,Y 640.735,Z 417.38,A -85,B 0,C 180,E1 30023.851,E2 30023.851} C_VEL
LIN {X 0,Y 640.757,Z 417.41,A -85,B 0,C 180,E1 30020.687,E2 30020.687} C_VEL
LIN {X 0,Y 640.731,Z 417.391,A -85,B 0,C 180,E1 30018.093,E2 30018.093} C_VEL
LIN {X 0,Y 640.812,Z 417.383,A -85,B 0,C 180,E1 30015.148,E2 30015.148} C_VEL
LIN {X 0,Y 640.754,Z 417.382,A -85,B 0,C 180,E1 30014.479,E2 30014.479} C_VEL
LIN {X 0,Y 639.684,Z 417.617,A -85,B 0,C 180,E1 30014.011,E2 30014.011} C_VEL
LIN {X 0,Y 633.474,Z 418.314,A -85,B 0,C 180,E1 30012.825,E2 30012.825} C_VEL
LIN {X 0,Y 632.854,Z 418.648,A -85,B 0,C 180,E1 30012.443,E2 30012.443} C_VEL
LIN {X 0,Y 639.989,Z 436.415,A -85,B 0,C 180,E1 30010.302,E2 30010.302} C_VEL
LIN {X 0,Y 647.718,Z 456.763,A -85,B 0,C 180,E1 30008.046,E2 30008.046} C_VEL
LIN {X 0,Y 645.454,Z 496.579,A -85,B 0,C 180,E1 30005.043,E2 30005.043} C_VEL
LIN {X 0,Y 651.26,Z 524.251,A -85,B 0,C 180,E1 30004.276,E2 30004.276} C_VEL
LIN {X 0,Y 648.066,Z 777.216,A -85,B 0,C 180,E1 30001.198,E2 30001.198} C_VEL
LIN {X 0,Y 647.059,Z 847.675,A -85,B 0,C 180,E1 30000.318,E2 30000.318} C_VEL
LIN {X 0,Y 646.289,Z 870.599,A -85,B 0,C 180,E1 29999.876,E2 29999.876} C_VEL
LIN {X 0,Y 645.353,Z 892.031,A -85,B 0,C 180,E1 29999.321,E2 29999.321} C_VEL
LIN {X 0,Y 644.204,Z 913.173,A -85,B 0,C 180,E1 29998.609,E2 29998.609} C_VEL
LIN {X 0,Y 642.949,Z 933.972,A -85,B 0,C 180,E1 29997.762,E2 29997.762} C_VEL
LIN {X 0,Y 641.508,Z 954.757,A -85,B 0,C 180,E1 29996.733,E2 29996.733} C_VEL
LIN {X 0,Y 640.108,Z 974.513,A -85,B 0,C 180,E1 29995.589,E2 29995.589} C_VEL
LIN {X 0,Y 638.586,Z 994.566,A -85,B 0,C 180,E1 29994.22,E2 29994.22} C_VEL
LIN {X 0,Y 637.189,Z 1014.239,A -85,B 0,C 180,E1 29992.675,E2 29992.675} C_VEL
LIN {X 0,Y 636.021,Z 1031.19,A -85,B 0,C 180,E1 29991.149,E2 29991.149} C_VEL
LIN {X 0,Y 634.974,Z 1046.92,A -85,B 0,C 180,E1 29989.502,E2 29989.502} C_VEL
LIN {X 0,Y 634.082,Z 1061.801,A -85,B 0,C 180,E1 29987.719,E2 29987.719} C_VEL
LIN {X 0,Y 633.363,Z 1074.538,A -85,B 0,C 180,E1 29985.944,E2 29985.944} C_VEL
LIN {X 0,Y 632.8,Z 1086.571,A -85,B 0,C 180,E1 29983.99,E2 29983.99} C_VEL
LIN {X 0,Y 632.428,Z 1096.253,A -85,B 0,C 180,E1 29982.139,E2 29982.139} C_VEL
LIN {X 0,Y 632.158,Z 1105.022,A -85,B 0,C 180,E1 29980.112,E2 29980.112} C_VEL
LIN {X 0,Y 632.024,Z 1111.819,A -85,B 0,C 180,E1 29978.186,E2 29978.186} C_VEL
LIN {X 0,Y 631.944,Z 1117.448,A -85,B 0,C 180,E1 29976.085,E2 29976.085} C_VEL
LIN {X 0,Y 631.912,Z 1121.487,A -85,B 0,C 180,E1 29973.992,E2 29973.992} C_VEL
LIN {X 0,Y 631.907,Z 1123.722,A -85,B 0,C 180,E1 29971.904,E2 29971.904} C_VEL
LIN {X 0,Y 631.905,Z 1124.47,A -85,B 0,C 180,E1 29969.819,E2 29969.819} C_VEL
LIN {X 0,Y 631.904,Z 1123.588,A -85,B 0,C 180,E1 29967.824,E2 29967.824} C_VEL
LIN {X 0,Y 631.912,Z 1121.175,A -85,B 0,C 180,E1 29965.735,E2 29965.735} C_VEL
LIN {X 0,Y 631.947,Z 1117.445,A -85,B 0,C 180,E1 29963.823,E2 29963.823} C_VEL
LIN {X 0,Y 632.029,Z 1111.812,A -85,B 0,C 180,E1 29961.723,E2 29961.723} C_VEL
LIN {X 0,Y 632.159,Z 1105.013,A -85,B 0,C 180,E1 29959.796,E2 29959.796} C_VEL
LIN {X 0,Y 632.44,Z 1095.929,A -85,B 0,C 180,E1 29957.706,E2 29957.706} C_VEL
LIN {X 0,Y 632.802,Z 1086.553,A -85,B 0,C 180,E1 29955.916,E2 29955.916} C_VEL
LIN {X 0,Y 633.365,Z 1074.513,A -85,B 0,C 180,E1 29953.962,E2 29953.962} C_VEL
LIN {X 0,Y 634.081,Z 1061.765,A -85,B 0,C 180,E1 29952.186,E2 29952.186} C_VEL
LIN {X 0,Y 634.977,Z 1046.869,A -85,B 0,C 180,E1 29950.403,E2 29950.403} C_VEL
LIN {X 0,Y 635.998,Z 1031.554,A -85,B 0,C 180,E1 29948.796,E2 29948.796} C_VEL
LIN {X 0,Y 637.184,Z 1014.336,A -85,B 0,C 180,E1 29947.243,E2 29947.243} C_VEL
LIN {X 0,Y 638.55,Z 995.042,A -85,B 0,C 180,E1 29945.725,E2 29945.725} C_VEL
LIN {X 0,Y 640.003,Z 975.815,A -85,B 0,C 180,E1 29944.406,E2 29944.406} C_VEL
LIN {X 0,Y 641.446,Z 955.635,A -85,B 0,C 180,E1 29943.224,E2 29943.224} C_VEL
LIN {X 0,Y 642.898,Z 934.861,A -85,B 0,C 180,E1 29942.187,E2 29942.187} C_VEL
LIN {X 0,Y 644.2,Z 913.264,A -85,B 0,C 180,E1 29941.304,E2 29941.304} C_VEL
LIN {X 0,Y 645.414,Z 890.663,A -85,B 0,C 180,E1 29940.551,E2 29940.551} C_VEL
LIN {X 0,Y 646.324,Z 869.872,A -85,B 0,C 180,E1 29940.017,E2 29940.017} C_VEL
LIN {X 0,Y 647.082,Z 846.256,A -85,B 0,C 180,E1 29939.571,E2 29939.571} C_VEL
LIN {X 0,Y 649.354,Z 677.318,A -85,B 0,C 180,E1 29937.495,E2 29937.495} C_VEL
LIN {X 0,Y 651.123,Z 523.165,A -85,B 0,C 180,E1 29935.611,E2 29935.611} C_VEL
LIN {X 0,Y 645.433,Z 496.483,A -85,B 0,C 180,E1 29934.864,E2 29934.864} C_VEL
LIN {X 0,Y 647.72,Z 456.81,A -85,B 0,C 180,E1 29931.867,E2 29931.867} C_VEL
LIN {X 0,Y 640.405,Z 437.497,A -85,B 0,C 180,E1 29929.729,E2 29929.729} C_VEL
LIN {X 0,Y 634.163,Z 421.984,A -85,B 0,C 180,E1 29927.896,E2 29927.896} C_VEL
LIN {X 0,Y 632.857,Z 418.552,A -85,B 0,C 180,E1 29927.433,E2 29927.433} C_VEL
LIN {X 0,Y 632.822,Z 418.387,A -85,B 0,C 180,E1 29924.294,E2 29924.294} C_VEL
LIN {X 0,Y 632.806,Z 418.372,A -85,B 0,C 180,E1 29921.578,E2 29921.578} C_VEL
LIN {X 0,Y 632.848,Z 418.401,A -85,B 0,C 180,E1 29918.5,E2 29918.5} C_VEL
LIN {X 0,Y 632.792,Z 418.368,A -85,B 0,C 180,E1 29915.667,E2 29915.667} C_VEL
LIN {X 0,Y 632.874,Z 418.398,A -85,B 0,C 180,E1 29912.637,E2 29912.637} C_VEL
LIN {X 0,Y 632.789,Z 418.404,A -85,B 0,C 180,E1 29909.747,E2 29909.747} C_VEL
LIN {X 0,Y 632.826,Z 418.399,A -85,B 0,C 180,E1 29906.967,E2 29906.967} C_VEL
LIN {X 0,Y 632.796,Z 418.401,A -85,B 0,C 180,E1 29903.81,E2 29903.81} C_VEL
LIN {X 0,Y 632.801,Z 418.399,A -85,B 0,C 180,E1 29901.209,E2 29901.209} C_VEL
LIN {X 0,Y 632.831,Z 418.396,A -85,B 0,C 180,E1 29898.04,E2 29898.04} C_VEL
LIN {X 0,Y 632.803,Z 418.4,A -85,B 0,C 180,E1 29895.3,E2 29895.3} C_VEL
LIN {X 0,Y 632.883,Z 418.386,A -85,B 0,C 180,E1 29892.315,E2 29892.315} C_VEL
LIN {X 0,Y 632.807,Z 418.398,A -85,B 0,C 180,E1 29889.367,E2 29889.367} C_VEL
LIN {X 0,Y 632.862,Z 418.395,A -85,B 0,C 180,E1 29886.532,E2 29886.532} C_VEL
LIN {X 0,Y 632.818,Z 418.388,A -85,B 0,C 180,E1 29883.442,E2 29883.442} C_VEL
LIN {X 0,Y 632.845,Z 418.401,A -85,B 0,C 180,E1 29880.634,E2 29880.634} C_VEL
LIN {X 0,Y 632.835,Z 418.397,A -85,B 0,C 180,E1 29877.464,E2 29877.464} C_VEL
LIN {X 0,Y 632.841,Z 418.39,A -85,B 0,C 180,E1 29874.651,E2 29874.651} C_VEL
LIN {X 0,Y 632.841,Z 418.393,A -85,B 0,C 180,E1 29871.367,E2 29871.367} C_VEL
LIN {X 0,Y 632.851,Z 418.396,A -85,B 0,C 180,E1 29868.517,E2 29868.517} C_VEL
LIN {X 0,Y 632.847,Z 418.389,A -85,B 0,C 180,E1 29865.263,E2 29865.263} C_VEL
LIN {X 0,Y 632.868,Z 418.391,A -85,B 0,C 180,E1 29862.309,E2 29862.309} C_VEL
LIN {X 0,Y 632.854,Z 418.393,A -85,B 0,C 180,E1 29859.176,E2 29859.176} C_VEL
LIN {X 0,Y 632.876,Z 418.397,A -85,B 0,C 180,E1 29856.174,E2 29856.174} C_VEL
LIN {X 0,Y 632.857,Z 418.394,A -85,B 0,C 180,E1 29853.012,E2 29853.012} C_VEL
LIN {X 0,Y 632.895,Z 418.391,A -85,B 0,C 180,E1 29849.946,E2 29849.946} C_VEL
LIN {X 0,Y 632.853,Z 418.368,A -85,B 0,C 180,E1 29846.753,E2 29846.753} C_VEL
LIN {X 0,Y 632.89,Z 418.399,A -85,B 0,C 180,E1 29843.668,E2 29843.668} C_VEL
LIN {X 0,Y 632.852,Z 418.362,A -85,B 0,C 180,E1 29840.569,E2 29840.569} C_VEL
LIN {X 0,Y 632.887,Z 418.384,A -85,B 0,C 180,E1 29837.545,E2 29837.545} C_VEL
LIN {X 0,Y 632.865,Z 418.396,A -85,B 0,C 180,E1 29834.421,E2 29834.421} C_VEL
LIN {X 0,Y 632.93,Z 418.692,A -85,B 0,C 180,E1 29833.265,E2 29833.265} C_VEL
LIN {X 0,Y 641.843,Z 440.26,A -85,B 0,C 180,E1 29830.789,E2 29830.789} C_VEL
LIN {X 0,Y 647.828,Z 455.349,A -85,B 0,C 180,E1 29829.212,E2 29829.212} C_VEL
LIN {X 0,Y 649.8,Z 459.28,A -85,B 0,C 180,E1 29829.015,E2 29829.015} C_VEL
LIN {X 0,Y 654.267,Z 480.517,A -85,B 0,C 180,E1 29828.428,E2 29828.428} C_VEL
LIN {X 0,Y 650.848,Z 727.916,A -85,B 0,C 180,E1 29825.332,E2 29825.332} C_VEL
LIN {X 0,Y 649.351,Z 844.334,A -85,B 0,C 180,E1 29823.885,E2 29823.885} C_VEL
LIN {X 0,Y 648.544,Z 869.791,A -85,B 0,C 180,E1 29823.411,E2 29823.411} C_VEL
LIN {X 0,Y 647.682,Z 890.807,A -85,B 0,C 180,E1 29822.89,E2 29822.89} C_VEL
LIN {X 0,Y 646.447,Z 916.237,A -85,B 0,C 180,E1 29822.087,E2 29822.087} C_VEL
LIN {X 0,Y 645.264,Z 937.213,A -85,B 0,C 180,E1 29821.273,E2 29821.273} C_VEL
LIN {X 0,Y 643.809,Z 961.261,A -85,B 0,C 180,E1 29820.16,E2 29820.16} C_VEL
LIN {X 0,Y 642.53,Z 979.891,A -85,B 0,C 180,E1 29819.149,E2 29819.149} C_VEL
LIN {X 0,Y 641,Z 1000.154,A -85,B 0,C 180,E1 29817.868,E2 29817.868} C_VEL
LIN {X 0,Y 639.428,Z 1019.818,A -85,B 0,C 180,E1 29816.416,E2 29816.416} C_VEL
LIN {X 0,Y 637.991,Z 1038.165,A -85,B 0,C 180,E1 29814.886,E2 29814.886} C_VEL
LIN {X 0,Y 636.645,Z 1055.525,A -85,B 0,C 180,E1 29813.217,E2 29813.217} C_VEL
LIN {X 0,Y 635.556,Z 1070.507,A -85,B 0,C 180,E1 29811.597,E2 29811.597} C_VEL
LIN {X 0,Y 634.48,Z 1086.516,A -85,B 0,C 180,E1 29809.613,E2 29809.613} C_VEL
LIN {X 0,Y 633.672,Z 1099.785,A -85,B 0,C 180,E1 29807.731,E2 29807.731} C_VEL
LIN {X 0,Y 633.012,Z 1112.284,A -85,B 0,C 180,E1 29805.671,E2 29805.671} C_VEL
LIN {X 0,Y 632.586,Z 1122.019,A -85,B 0,C 180,E1 29803.809,E2 29803.809} C_VEL
LIN {X 0,Y 632.25,Z 1131.835,A -85,B 0,C 180,E1 29801.587,E2 29801.587} C_VEL
LIN {X 0,Y 632.076,Z 1138.816,A -85,B 0,C 180,E1 29799.653,E2 29799.653} C_VEL
LIN {X 0,Y 631.949,Z 1145.243,A -85,B 0,C 180,E1 29797.455,E2 29797.455} C_VEL
LIN {X 0,Y 631.902,Z 1149.655,A -85,B 0,C 180,E1 29795.357,E2 29795.357} C_VEL
LIN {X 0,Y 631.908,Z 1152.464,A -85,B 0,C 180,E1 29793.447,E2 29793.447} C_VEL
LIN {X 0,Y 631.909,Z 1154.214,A -85,B 0,C 180,E1 29791.179,E2 29791.179} C_VEL
LIN {X 0,Y 631.885,Z 1154.327,A -85,B 0,C 180,E1 29789.275,E2 29789.275} C_VEL
LIN {X 0,Y 631.886,Z 1153.224,A -85,B 0,C 180,E1 29787.279,E2 29787.279} C_VEL
LIN {X 0,Y 631.9,Z 1150.292,A -85,B 0,C 180,E1 29785.007,E2 29785.007} C_VEL
LIN {X 0,Y 631.952,Z 1146.689,A -85,B 0,C 180,E1 29783.185,E2 29783.185} C_VEL
LIN {X 0,Y 632.027,Z 1140.934,A -85,B 0,C 180,E1 29780.989,E2 29780.989} C_VEL
LIN {X 0,Y 632.188,Z 1133.602,A -85,B 0,C 180,E1 29778.874,E2 29778.874} C_VEL
LIN {X 0,Y 632.47,Z 1125.531,A -85,B 0,C 180,E1 29776.934,E2 29776.934} C_VEL
LIN {X 0,Y 632.906,Z 1114.861,A -85,B 0,C 180,E1 29774.796,E2 29774.796} C_VEL
LIN {X 0,Y 633.444,Z 1103.97,A -85,B 0,C 180,E1 29772.926,E2 29772.926} C_VEL
LIN {X 0,Y 634.274,Z 1089.478,A -85,B 0,C 180,E1 29770.785,E2 29770.785} C_VEL
LIN {X 0,Y 635.169,Z 1076.076,A -85,B 0,C 180,E1 29769.063,E2 29769.063} C_VEL
LIN {X 0,Y 636.439,Z 1058.302,A -85,B 0,C 180,E1 29767.069,E2 29767.069} C_VEL
LIN {X 0,Y 637.623,Z 1042.795,A -85,B 0,C 180,E1 29765.544,E2 29765.544} C_VEL
LIN {X 0,Y 639.184,Z 1022.857,A -85,B 0,C 180,E1 29763.823,E2 29763.823} C_VEL
LIN {X 0,Y 640.54,Z 1005.72,A -85,B 0,C 180,E1 29762.53,E2 29762.53} C_VEL
LIN {X 0,Y 642.174,Z 984.779,A -85,B 0,C 180,E1 29761.139,E2 29761.139} C_VEL
LIN {X 0,Y 643.47,Z 965.886,A -85,B 0,C 180,E1 29760.079,E2 29760.079} C_VEL
LIN {X 0,Y 644.899,Z 944.214,A -85,B 0,C 180,E1 29759.027,E2 29759.027} C_VEL
LIN {X 0,Y 646.181,Z 921.337,A -85,B 0,C 180,E1 29758.1,E2 29758.1} C_VEL
LIN {X 0,Y 647.223,Z 900.67,A -85,B 0,C 180,E1 29757.399,E2 29757.399} C_VEL
LIN {X 0,Y 648.322,Z 874.941,A -85,B 0,C 180,E1 29756.704,E2 29756.704} C_VEL
LIN {X 0,Y 649.079,Z 853.654,A -85,B 0,C 180,E1 29756.271,E2 29756.271} C_VEL
LIN {X 0,Y 649.665,Z 826.232,A -85,B 0,C 180,E1 29755.872,E2 29755.872} C_VEL
LIN {X 0,Y 652.504,Z 598.11,A -85,B 0,C 180,E1 29753.058,E2 29753.058} C_VEL
LIN {X 0,Y 654.106,Z 478.918,A -85,B 0,C 180,E1 29751.541,E2 29751.541} C_VEL
LIN {X 0,Y 649.35,Z 458.044,A -85,B 0,C 180,E1 29750.938,E2 29750.938} C_VEL
LIN {X 0,Y 647.548,Z 454.805,A -85,B 0,C 180,E1 29750.749,E2 29750.749} C_VEL
LIN {X 0,Y 639.565,Z 434.739,A -85,B 0,C 180,E1 29748.6,E2 29748.6} C_VEL
LIN {X 0,Y 632.914,Z 418.598,A -85,B 0,C 180,E1 29746.714,E2 29746.714} C_VEL
LIN {X 0,Y 632.86,Z 418.365,A -85,B 0,C 180,E1 29743.645,E2 29743.645} C_VEL
LIN {X 0,Y 632.886,Z 418.377,A -85,B 0,C 180,E1 29740.611,E2 29740.611} C_VEL
LIN {X 0,Y 632.858,Z 418.394,A -85,B 0,C 180,E1 29737.58,E2 29737.58} C_VEL
LIN {X 0,Y 632.887,Z 418.363,A -85,B 0,C 180,E1 29734.554,E2 29734.554} C_VEL
LIN {X 0,Y 632.854,Z 418.399,A -85,B 0,C 180,E1 29731.426,E2 29731.426} C_VEL
LIN {X 0,Y 632.895,Z 418.387,A -85,B 0,C 180,E1 29728.359,E2 29728.359} C_VEL
LIN {X 0,Y 632.848,Z 418.394,A -85,B 0,C 180,E1 29725.252,E2 29725.252} C_VEL
LIN {X 0,Y 632.894,Z 418.385,A -85,B 0,C 180,E1 29722.185,E2 29722.185} C_VEL
LIN {X 0,Y 632.841,Z 418.39,A -85,B 0,C 180,E1 29719.118,E2 29719.118} C_VEL
LIN {X 0,Y 632.896,Z 418.396,A -85,B 0,C 180,E1 29716.05,E2 29716.05} C_VEL
LIN {X 0,Y 632.834,Z 418.396,A -85,B 0,C 180,E1 29713.058,E2 29713.058} C_VEL
LIN {X 0,Y 632.894,Z 418.385,A -85,B 0,C 180,E1 29710.008,E2 29710.008} C_VEL
LIN {X 0,Y 632.829,Z 418.396,A -85,B 0,C 180,E1 29706.988,E2 29706.988} C_VEL
LIN {X 0,Y 632.891,Z 418.389,A -85,B 0,C 180,E1 29703.986,E2 29703.986} C_VEL
LIN {X 0,Y 632.824,Z 418.387,A -85,B 0,C 180,E1 29700.996,E2 29700.996} C_VEL
LIN {X 0,Y 632.857,Z 418.397,A -85,B 0,C 180,E1 29698.189,E2 29698.189} C_VEL
LIN {X 0,Y 632.825,Z 418.399,A -85,B 0,C 180,E1 29695.015,E2 29695.015} C_VEL
LIN {X 0,Y 632.831,Z 418.392,A -85,B 0,C 180,E1 29692.282,E2 29692.282} C_VEL
LIN {X 0,Y 632.83,Z 418.398,A -85,B 0,C 180,E1 29689.07,E2 29689.07} C_VEL
LIN {X 0,Y 632.814,Z 418.396,A -85,B 0,C 180,E1 29686.348,E2 29686.348} C_VEL
LIN {X 0,Y 632.86,Z 418.389,A -85,B 0,C 180,E1 29683.288,E2 29683.288} C_VEL
LIN {X 0,Y 632.802,Z 418.4,A -85,B 0,C 180,E1 29680.428,E2 29680.428} C_VEL
LIN {X 0,Y 632.889,Z 418.397,A -85,B 0,C 180,E1 29677.424,E2 29677.424} C_VEL
LIN {X 0,Y 632.795,Z 418.401,A -85,B 0,C 180,E1 29674.445,E2 29674.445} C_VEL
LIN {X 0,Y 632.845,Z 418.392,A -85,B 0,C 180,E1 29671.603,E2 29671.603} C_VEL
LIN {X 0,Y 632.795,Z 418.396,A -85,B 0,C 180,E1 29668.569,E2 29668.569} C_VEL
LIN {X 0,Y 632.799,Z 418.402,A -85,B 0,C 180,E1 29665.879,E2 29665.879} C_VEL
LIN {X 0,Y 632.808,Z 418.386,A -85,B 0,C 180,E1 29662.635,E2 29662.635} C_VEL
LIN {X 0,Y 632.792,Z 418.393,A -85,B 0,C 180,E1 29660.029,E2 29660.029} C_VEL
LIN {X 0,Y 632.873,Z 418.393,A -85,B 0,C 180,E1 29657.013,E2 29657.013} C_VEL
LIN {X 0,Y 632.797,Z 418.372,A -85,B 0,C 180,E1 29654.032,E2 29654.032} C_VEL
LIN {X 0,Y 632.854,Z 418.648,A -85,B 0,C 180,E1 29652.443,E2 29652.443} C_VEL
LIN {X 0,Y 632.966,Z 425.815,A -85,B 0,C 180,E1 29651.773,E2 29651.773} C_VEL
LIN {X 0,Y 632.976,Z 437.521,A -85,B 0,C 180,E1 29650.777,E2 29650.777} C_VEL
LIN {X 0,Y 634.514,Z 443.371,A -85,B 0,C 180,E1 29650.133,E2 29650.133} C_VEL
LIN {X 0,Y 640.752,Z 459.941,A -85,B 0,C 180,E1 29648.281,E2 29648.281} C_VEL
LIN {X 0,Y 638.602,Z 496.629,A -85,B 0,C 180,E1 29645.492,E2 29645.492} C_VEL
LIN {X 0,Y 644.8,Z 525.803,A -85,B 0,C 180,E1 29644.68,E2 29644.68} C_VEL
LIN {X 0,Y 641.384,Z 783.662,A -85,B 0,C 180,E1 29641.524,E2 29641.524} C_VEL
LIN {X 0,Y 640.401,Z 848.148,A -85,B 0,C 180,E1 29640.711,E2 29640.711} C_VEL
LIN {X 0,Y 639.586,Z 870.917,A -85,B 0,C 180,E1 29640.267,E2 29640.267} C_VEL
LIN {X 0,Y 638.596,Z 892.346,A -85,B 0,C 180,E1 29639.707,E2 29639.707} C_VEL
LIN {X 0,Y 637.369,Z 913.304,A -85,B 0,C 180,E1 29638.996,E2 29638.996} C_VEL
LIN {X 0,Y 635.992,Z 934.671,A -85,B 0,C 180,E1 29638.116,E2 29638.116} C_VEL
LIN {X 0,Y 634.419,Z 955.531,A -85,B 0,C 180,E1 29637.066,E2 29637.066} C_VEL
LIN {X 0,Y 632.826,Z 976.013,A -85,B 0,C 180,E1 29635.855,E2 29635.855} C_VEL
LIN {X 0,Y 631.357,Z 993.918,A -85,B 0,C 180,E1 29634.615,E2 29634.615} C_VEL
LIN {X 0,Y 629.752,Z 1013.492,A -85,B 0,C 180,E1 29633.047,E2 29633.047} C_VEL
LIN {X 0,Y 628.344,Z 1031.685,A -85,B 0,C 180,E1 29631.371,E2 29631.371} C_VEL
LIN {X 0,Y 627.248,Z 1046.924,A -85,B 0,C 180,E1 29629.752,E2 29629.752} C_VEL
LIN {X 0,Y 626.275,Z 1061.804,A -85,B 0,C 180,E1 29627.947,E2 29627.947} C_VEL
LIN {X 0,Y 625.502,Z 1074.54,A -85,B 0,C 180,E1 29626.15,E2 29626.15} C_VEL
LIN {X 0,Y 624.881,Z 1086.721,A -85,B 0,C 180,E1 29624.144,E2 29624.144} C_VEL
LIN {X 0,Y 624.482,Z 1096.255,A -85,B 0,C 180,E1 29622.296,E2 29622.296} C_VEL
LIN {X 0,Y 624.188,Z 1105.024,A -85,B 0,C 180,E1 29620.242,E2 29620.242} C_VEL
LIN {X 0,Y 624.044,Z 1111.821,A -85,B 0,C 180,E1 29618.291,E2 29618.291} C_VEL
LIN {X 0,Y 623.95,Z 1117.449,A -85,B 0,C 180,E1 29616.164,E2 29616.164} C_VEL
LIN {X 0,Y 623.914,Z 1121.487,A -85,B 0,C 180,E1 29614.044,E2 29614.044} C_VEL
LIN {X 0,Y 623.907,Z 1123.722,A -85,B 0,C 180,E1 29611.929,E2 29611.929} C_VEL
LIN {X 0,Y 623.904,Z 1124.47,A -85,B 0,C 180,E1 29609.816,E2 29609.816} C_VEL
LIN {X 0,Y 623.903,Z 1123.588,A -85,B 0,C 180,E1 29607.796,E2 29607.796} C_VEL
LIN {X 0,Y 623.91,Z 1121.175,A -85,B 0,C 180,E1 29605.68,E2 29605.68} C_VEL
LIN {X 0,Y 623.951,Z 1117.444,A -85,B 0,C 180,E1 29603.744,E2 29603.744} C_VEL
LIN {X 0,Y 624.043,Z 1111.811,A -85,B 0,C 180,E1 29601.616,E2 29601.616} C_VEL
LIN {X 0,Y 624.19,Z 1105.011,A -85,B 0,C 180,E1 29599.664,E2 29599.664} C_VEL
LIN {X 0,Y 624.483,Z 1096.232,A -85,B 0,C 180,E1 29597.609,E2 29597.609} C_VEL
LIN {X 0,Y 624.89,Z 1086.549,A -85,B 0,C 180,E1 29595.734,E2 29595.734} C_VEL
LIN {X 0,Y 625.542,Z 1073.871,A -85,B 0,C 180,E1 29593.661,E2 29593.661} C_VEL
LIN {X 0,Y 626.323,Z 1061.056,A -85,B 0,C 180,E1 29591.862,E2 29591.862} C_VEL
LIN {X 0,Y 627.261,Z 1046.724,A -85,B 0,C 180,E1 29590.136,E2 29590.136} C_VEL
LIN {X 0,Y 628.423,Z 1030.622,A -85,B 0,C 180,E1 29588.436,E2 29588.436} C_VEL
LIN {X 0,Y 629.91,Z 1011.548,A -85,B 0,C 180,E1 29586.692,E2 29586.692} C_VEL
LIN {X 0,Y 631.42,Z 993.134,A -85,B 0,C 180,E1 29585.238,E2 29585.238} C_VEL
LIN {X 0,Y 632.966,Z 974.43,A -85,B 0,C 180,E1 29583.95,E2 29583.95} C_VEL
LIN {X 0,Y 634.479,Z 954.804,A -85,B 0,C 180,E1 29582.805,E2 29582.805} C_VEL
LIN {X 0,Y 636.039,Z 933.856,A -85,B 0,C 180,E1 29581.758,E2 29581.758} C_VEL
LIN {X 0,Y 637.391,Z 912.988,A -85,B 0,C 180,E1 29580.901,E2 29580.901} C_VEL
LIN {X 0,Y 638.73,Z 889.583,A -85,B 0,C 180,E1 29580.125,E2 29580.125} C_VEL
LIN {X 0,Y 639.656,Z 869.36,A -85,B 0,C 180,E1 29579.607,E2 29579.607} C_VEL
LIN {X 0,Y 640.446,Z 845.367,A -85,B 0,C 180,E1 29579.158,E2 29579.158} C_VEL
LIN {X 0,Y 643.004,Z 660.681,A -85,B 0,C 180,E1 29576.881,E2 29576.881} C_VEL
LIN {X 0,Y 644.635,Z 524.589,A -85,B 0,C 180,E1 29575.203,E2 29575.203} C_VEL
LIN {X 0,Y 638.561,Z 496.132,A -85,B 0,C 180,E1 29574.393,E2 29574.393} C_VEL
LIN {X 0,Y 640.784,Z 460.05,A -85,B 0,C 180,E1 29571.639,E2 29571.639} C_VEL
LIN {X 0,Y 633.113,Z 439.867,A -85,B 0,C 180,E1 29569.365,E2 29569.365} C_VEL
LIN {X 0,Y 625.933,Z 422.413,A -85,B 0,C 180,E1 29567.241,E2 29567.241} C_VEL
LIN {X 0,Y 624.968,Z 419.548,A -85,B 0,C 180,E1 29566.85,E2 29566.85} C_VEL
LIN {X 0,Y 624.869,Z 419.388,A -85,B 0,C 180,E1 29563.939,E2 29563.939} C_VEL
LIN {X 0,Y 624.935,Z 419.349,A -85,B 0,C 180,E1 29560.957,E2 29560.957} C_VEL
LIN {X 0,Y 624.866,Z 419.39,A -85,B 0,C 180,E1 29558.03,E2 29558.03} C_VEL
LIN {X 0,Y 624.873,Z 419.357,A -85,B 0,C 180,E1 29555.286,E2 29555.286} C_VEL
LIN {X 0,Y 624.869,Z 419.385,A -85,B 0,C 180,E1 29552.09,E2 29552.09} C_VEL
LIN {X 0,Y 624.854,Z 419.394,A -85,B 0,C 180,E1 29549.424,E2 29549.424} C_VEL
LIN {X 0,Y 624.9,Z 419.391,A -85,B 0,C 180,E1 29546.31,E2 29546.31} C_VEL
LIN {X 0,Y 624.852,Z 419.39,A -85,B 0,C 180,E1 29543.481,E2 29543.481} C_VEL
LIN {X 0,Y 624.938,Z 419.376,A -85,B 0,C 180,E1 29540.512,E2 29540.512} C_VEL
LIN {X 0,Y 624.859,Z 419.385,A -85,B 0,C 180,E1 29537.5,E2 29537.5} C_VEL
LIN {X 0,Y 624.936,Z 419.39,A -85,B 0,C 180,E1 29534.534,E2 29534.534} C_VEL
LIN {X 0,Y 624.867,Z 419.386,A -85,B 0,C 180,E1 29531.445,E2 29531.445} C_VEL
LIN {X 0,Y 624.921,Z 419.378,A -85,B 0,C 180,E1 29528.558,E2 29528.558} C_VEL
LIN {X 0,Y 624.881,Z 419.387,A -85,B 0,C 180,E1 29525.509,E2 29525.509} C_VEL
LIN {X 0,Y 624.895,Z 419.379,A -85,B 0,C 180,E1 29522.751,E2 29522.751} C_VEL
LIN {X 0,Y 624.894,Z 419.374,A -85,B 0,C 180,E1 29519.542,E2 29519.542} C_VEL
LIN {X 0,Y 624.899,Z 419.389,A -85,B 0,C 180,E1 29516.698,E2 29516.698} C_VEL
LIN {X 0,Y 624.905,Z 419.384,A -85,B 0,C 180,E1 29513.477,E2 29513.477} C_VEL
LIN {X 0,Y 624.898,Z 419.383,A -85,B 0,C 180,E1 29510.7,E2 29510.7} C_VEL
LIN {X 0,Y 624.926,Z 419.382,A -85,B 0,C 180,E1 29507.526,E2 29507.526} C_VEL
LIN {X 0,Y 624.904,Z 419.382,A -85,B 0,C 180,E1 29504.597,E2 29504.597} C_VEL
LIN {X 0,Y 624.933,Z 419.375,A -85,B 0,C 180,E1 29501.434,E2 29501.434} C_VEL
LIN {X 0,Y 624.917,Z 419.382,A -85,B 0,C 180,E1 29498.407,E2 29498.407} C_VEL
LIN {X 0,Y 624.92,Z 419.38,A -85,B 0,C 180,E1 29495.114,E2 29495.114} C_VEL
LIN {X 0,Y 624.95,Z 419.385,A -85,B 0,C 180,E1 29492.028,E2 29492.028} C_VEL
LIN {X 0,Y 624.919,Z 419.386,A -85,B 0,C 180,E1 29488.873,E2 29488.873} C_VEL
LIN {X 0,Y 624.948,Z 419.345,A -85,B 0,C 180,E1 29485.81,E2 29485.81} C_VEL
LIN {X 0,Y 624.92,Z 419.387,A -85,B 0,C 180,E1 29482.669,E2 29482.669} C_VEL
LIN {X 0,Y 624.946,Z 419.358,A -85,B 0,C 180,E1 29479.604,E2 29479.604} C_VEL
LIN {X 0,Y 624.921,Z 419.353,A -85,B 0,C 180,E1 29476.527,E2 29476.527} C_VEL
LIN {X 0,Y 624.975,Z 419.595,A -85,B 0,C 180,E1 29473.877,E2 29473.877} C_VEL
LIN {X 0,Y 633.901,Z 441.037,A -85,B 0,C 180,E1 29471.338,E2 29471.338} C_VEL
LIN {X 0,Y 639.77,Z 455.787,A -85,B 0,C 180,E1 29469.758,E2 29469.758} C_VEL
LIN {X 0,Y 643.872,Z 463.173,A -85,B 0,C 180,E1 29469.36,E2 29469.36} C_VEL
LIN {X 0,Y 647.806,Z 482.235,A -85,B 0,C 180,E1 29468.828,E2 29468.828} C_VEL
LIN {X 0,Y 644.071,Z 729.168,A -85,B 0,C 180,E1 29465.698,E2 29465.698} C_VEL
LIN {X 0,Y 642.449,Z 844.256,A -85,B 0,C 180,E1 29464.248,E2 29464.248} C_VEL
LIN {X 0,Y 641.59,Z 869.776,A -85,B 0,C 180,E1 29463.768,E2 29463.768} C_VEL
LIN {X 0,Y 640.676,Z 890.666,A -85,B 0,C 180,E1 29463.244,E2 29463.244} C_VEL
LIN {X 0,Y 639.413,Z 915.279,A -85,B 0,C 180,E1 29462.464,E2 29462.464} C_VEL
LIN {X 0,Y 638.153,Z 935.921,A -85,B 0,C 180,E1 29461.661,E2 29461.661} C_VEL
LIN {X 0,Y 636.744,Z 958.545,A -85,B 0,C 180,E1 29460.623,E2 29460.623} C_VEL
LIN {X 0,Y 635.216,Z 979.449,A -85,B 0,C 180,E1 29459.486,E2 29459.486} C_VEL
LIN {X 0,Y 633.675,Z 1000.082,A -85,B 0,C 180,E1 29458.203,E2 29458.203} C_VEL
LIN {X 0,Y 632.181,Z 1018.323,A -85,B 0,C 180,E1 29456.867,E2 29456.867} C_VEL
LIN {X 0,Y 630.791,Z 1034.836,A -85,B 0,C 180,E1 29455.491,E2 29455.491} C_VEL
LIN {X 0,Y 629.213,Z 1053.672,A -85,B 0,C 180,E1 29453.706,E2 29453.706} C_VEL
LIN {X 0,Y 628.018,Z 1068.777,A -85,B 0,C 180,E1 29452.07,E2 29452.07} C_VEL
LIN {X 0,Y 626.817,Z 1085.113,A -85,B 0,C 180,E1 29450.058,E2 29450.058} C_VEL
LIN {X 0,Y 625.946,Z 1097.878,A -85,B 0,C 180,E1 29448.246,E2 29448.246} C_VEL
LIN {X 0,Y 625.211,Z 1110.731,A -85,B 0,C 180,E1 29446.157,E2 29446.157} C_VEL
LIN {X 0,Y 624.701,Z 1121.1,A -85,B 0,C 180,E1 29444.175,E2 29444.175} C_VEL
LIN {X 0,Y 624.338,Z 1130.77,A -85,B 0,C 180,E1 29442.017,E2 29442.017} C_VEL
LIN {X 0,Y 624.1,Z 1138.21,A -85,B 0,C 180,E1 29439.964,E2 29439.964} C_VEL
LIN {X 0,Y 623.983,Z 1143.999,A -85,B 0,C 180,E1 29438.014,E2 29438.014} C_VEL
LIN {X 0,Y 623.924,Z 1149.175,A -85,B 0,C 180,E1 29435.702,E2 29435.702} C_VEL
LIN {X 0,Y 623.914,Z 1152.124,A -85,B 0,C 180,E1 29433.767,E2 29433.767} C_VEL
LIN {X 0,Y 623.898,Z 1154.103,A -85,B 0,C 180,E1 29431.561,E2 29431.561} C_VEL
LIN {X 0,Y 623.884,Z 1154.373,A -85,B 0,C 180,E1 29429.449,E2 29429.449} C_VEL
LIN {X 0,Y 623.899,Z 1153.428,A -85,B 0,C 180,E1 29427.52,E2 29427.52} C_VEL
LIN {X 0,Y 623.912,Z 1150.769,A -85,B 0,C 180,E1 29425.22,E2 29425.22} C_VEL
LIN {X 0,Y 623.954,Z 1146.895,A -85,B 0,C 180,E1 29423.189,E2 29423.189} C_VEL
LIN {X 0,Y 624.02,Z 1141.71,A -85,B 0,C 180,E1 29421.151,E2 29421.151} C_VEL
LIN {X 0,Y 624.201,Z 1134.308,A -85,B 0,C 180,E1 29418.917,E2 29418.917} C_VEL
LIN {X 0,Y 624.478,Z 1126.75,A -85,B 0,C 180,E1 29417.046,E2 29417.046} C_VEL
LIN {X 0,Y 624.935,Z 1116.404,A -85,B 0,C 180,E1 29414.882,E2 29414.882} C_VEL
LIN {X 0,Y 625.519,Z 1105.115,A -85,B 0,C 180,E1 29412.895,E2 29412.895} C_VEL
LIN {X 0,Y 626.332,Z 1092.119,A -85,B 0,C 180,E1 29410.897,E2 29410.897} C_VEL
LIN {X 0,Y 627.346,Z 1077.615,A -85,B 0,C 180,E1 29408.985,E2 29408.985} C_VEL
LIN {X 0,Y 628.564,Z 1061.998,A -85,B 0,C 180,E1 29407.161,E2 29407.161} C_VEL
LIN {X 0,Y 629.943,Z 1044.821,A -85,B 0,C 180,E1 29405.426,E2 29405.426} C_VEL
LIN {X 0,Y 631.502,Z 1026.495,A -85,B 0,C 180,E1 29403.784,E2 29403.784} C_VEL
LIN {X 0,Y 633.007,Z 1008.538,A -85,B 0,C 180,E1 29402.394,E2 29402.394} C_VEL
LIN {X 0,Y 634.421,Z 990.239,A -85,B 0,C 180,E1 29401.166,E2 29401.166} C_VEL
LIN {X 0,Y 636.078,Z 967.313,A -85,B 0,C 180,E1 29399.835,E2 29399.835} C_VEL
LIN {X 0,Y 637.425,Z 947.863,A -85,B 0,C 180,E1 29398.868,E2 29398.868} C_VEL
LIN {X 0,Y 638.943,Z 923.668,A -85,B 0,C 180,E1 29397.846,E2 29397.846} C_VEL
LIN {X 0,Y 640.065,Z 902.859,A -85,B 0,C 180,E1 29397.122,E2 29397.122} C_VEL
LIN {X 0,Y 641.192,Z 879.224,A -85,B 0,C 180,E1 29396.446,E2 29396.446} C_VEL
LIN {X 0,Y 642.083,Z 855.667,A -85,B 0,C 180,E1 29395.947,E2 29395.947} C_VEL
LIN {X 0,Y 642.729,Z 831.408,A -85,B 0,C 180,E1 29395.57,E2 29395.57} C_VEL
LIN {X 0,Y 645.895,Z 600.407,A -85,B 0,C 180,E1 29392.682,E2 29392.682} C_VEL
LIN {X 0,Y 647.642,Z 480.539,A -85,B 0,C 180,E1 29391.138,E2 29391.138} C_VEL
LIN {X 0,Y 643.461,Z 462.09,A -85,B 0,C 180,E1 29390.596,E2 29390.596} C_VEL
LIN {X 0,Y 639.548,Z 455.342,A -85,B 0,C 180,E1 29390.213,E2 29390.213} C_VEL
LIN {X 0,Y 631.029,Z 434.008,A -85,B 0,C 180,E1 29387.865,E2 29387.865} C_VEL
LIN {X 0,Y 624.976,Z 419.608,A -85,B 0,C 180,E1 29386.122,E2 29386.122} C_VEL
LIN {X 0,Y 624.941,Z 419.356,A -85,B 0,C 180,E1 29383.094,E2 29383.094} C_VEL
LIN {X 0,Y 624.932,Z 419.35,A -85,B 0,C 180,E1 29379.911,E2 29379.911} C_VEL
LIN {X 0,Y 624.953,Z 419.384,A -85,B 0,C 180,E1 29376.719,E2 29376.719} C_VEL
LIN {X 0,Y 624.913,Z 419.351,A -85,B 0,C 180,E1 29373.527,E2 29373.527} C_VEL
LIN {X 0,Y 624.953,Z 419.385,A -85,B 0,C 180,E1 29370.416,E2 29370.416} C_VEL
LIN {X 0,Y 624.911,Z 419.386,A -85,B 0,C 180,E1 29367.337,E2 29367.337} C_VEL
LIN {X 0,Y 624.956,Z 419.382,A -85,B 0,C 180,E1 29364.221,E2 29364.221} C_VEL
LIN {X 0,Y 624.906,Z 419.384,A -85,B 0,C 180,E1 29361.2,E2 29361.2} C_VEL
LIN {X 0,Y 624.953,Z 419.372,A -85,B 0,C 180,E1 29358.083,E2 29358.083} C_VEL
LIN {X 0,Y 624.899,Z 419.379,A -85,B 0,C 180,E1 29355.023,E2 29355.023} C_VEL
LIN {X 0,Y 624.954,Z 419.386,A -85,B 0,C 180,E1 29351.911,E2 29351.911} C_VEL
LIN {X 0,Y 624.894,Z 419.383,A -85,B 0,C 180,E1 29348.929,E2 29348.929} C_VEL
LIN {X 0,Y 624.955,Z 419.374,A -85,B 0,C 180,E1 29345.877,E2 29345.877} C_VEL
LIN {X 0,Y 624.887,Z 419.387,A -85,B 0,C 180,E1 29342.843,E2 29342.843} C_VEL
LIN {X 0,Y 624.959,Z 419.373,A -85,B 0,C 180,E1 29339.817,E2 29339.817} C_VEL
LIN {X 0,Y 624.88,Z 419.377,A -85,B 0,C 180,E1 29336.789,E2 29336.789} C_VEL
LIN {X 0,Y 624.957,Z 419.385,A -85,B 0,C 180,E1 29333.754,E2 29333.754} C_VEL
LIN {X 0,Y 624.875,Z 419.387,A -85,B 0,C 180,E1 29330.792,E2 29330.792} C_VEL
LIN {X 0,Y 624.922,Z 419.38,A -85,B 0,C 180,E1 29327.901,E2 29327.901} C_VEL
LIN {X 0,Y 624.872,Z 419.389,A -85,B 0,C 180,E1 29324.786,E2 29324.786} C_VEL
LIN {X 0,Y 624.89,Z 419.383,A -85,B 0,C 180,E1 29322.012,E2 29322.012} C_VEL
LIN {X 0,Y 624.871,Z 419.385,A -85,B 0,C 180,E1 29318.799,E2 29318.799} C_VEL
LIN {X 0,Y 624.862,Z 419.389,A -85,B 0,C 180,E1 29316.219,E2 29316.219} C_VEL
LIN {X 0,Y 624.918,Z 419.387,A -85,B 0,C 180,E1 29313.179,E2 29313.179} C_VEL
LIN {X 0,Y 624.851,Z 419.393,A -85,B 0,C 180,E1 29310.26,E2 29310.26} C_VEL
LIN {X 0,Y 624.931,Z 419.387,A -85,B 0,C 180,E1 29307.262,E2 29307.262} C_VEL
LIN {X 0,Y 624.845,Z 419.355,A -85,B 0,C 180,E1 29304.225,E2 29304.225} C_VEL
LIN {X 0,Y 624.943,Z 419.388,A -85,B 0,C 180,E1 29301.186,E2 29301.186} C_VEL
LIN {X 0,Y 624.853,Z 419.362,A -85,B 0,C 180,E1 29298.219,E2 29298.219} C_VEL
LIN {X 0,Y 624.904,Z 419.365,A -85,B 0,C 180,E1 29295.377,E2 29295.377} C_VEL
LIN {X 0,Y 624.973,Z 419.611,A -85,B 0,C 180,E1 29293.029,E2 29293.029} C_VEL
LIN {X 0,Y 633.412,Z 440.658,A -85,B 0,C 180,E1 29290.451,E2 29290.451} C_VEL
LIN {X 0,Y 634.514,Z 443.371,A -85,B 0,C 180,E1 29290.133,E2 29290.133} C_VEL
LIN {X 0,Y 635.635,Z 447.646,A -85,B 0,C 180,E1 29289.684,E2 29289.684} C_VEL
LIN {X 0,Y 635.58,Z 454.196,A -85,B 0,C 180,E1 29289.137,E2 29289.137} C_VEL
LIN {X 0,Y 633.388,Z 470.059,A -85,B 0,C 180,E1 29287.974,E2 29287.974} C_VEL
LIN {X 0,Y 631.781,Z 496.403,A -85,B 0,C 180,E1 29285.968,E2 29285.968} C_VEL
LIN {X 0,Y 638.361,Z 527.404,A -85,B 0,C 180,E1 29285.089,E2 29285.089} C_VEL
LIN {X 0,Y 634.785,Z 785.401,A -85,B 0,C 180,E1 29281.915,E2 29281.915} C_VEL
LIN {X 0,Y 633.794,Z 848.14,A -85,B 0,C 180,E1 29281.121,E2 29281.121} C_VEL
LIN {X 0,Y 632.946,Z 870.814,A -85,B 0,C 180,E1 29280.678,E2 29280.678} C_VEL
LIN {X 0,Y 631.946,Z 891.341,A -85,B 0,C 180,E1 29280.14,E2 29280.14} C_VEL
LIN {X 0,Y 630.571,Z 913.456,A -85,B 0,C 180,E1 29279.391,E2 29279.391} C_VEL
LIN {X 0,Y 629.063,Z 935.349,A -85,B 0,C 180,E1 29278.48,E2 29278.48} C_VEL
LIN {X 0,Y 627.397,Z 956.033,A -85,B 0,C 180,E1 29277.425,E2 29277.425} C_VEL
LIN {X 0,Y 625.7,Z 976.141,A -85,B 0,C 180,E1 29276.223,E2 29276.223} C_VEL
LIN {X 0,Y 624.111,Z 994.057,A -85,B 0,C 180,E1 29274.966,E2 29274.966} C_VEL
LIN {X 0,Y 622.361,Z 1013.644,A -85,B 0,C 180,E1 29273.38,E2 29273.38} C_VEL
LIN {X 0,Y 620.946,Z 1030.129,A -85,B 0,C 180,E1 29271.837,E2 29271.837} C_VEL
LIN {X 0,Y 619.549,Z 1047.036,A -85,B 0,C 180,E1 29270.008,E2 29270.008} C_VEL
LIN {X 0,Y 618.382,Z 1063.208,A -85,B 0,C 180,E1 29267.989,E2 29267.989} C_VEL
LIN {X 0,Y 617.575,Z 1075.814,A -85,B 0,C 180,E1 29266.17,E2 29266.17} C_VEL
LIN {X 0,Y 616.925,Z 1087.605,A -85,B 0,C 180,E1 29264.166,E2 29264.166} C_VEL
LIN {X 0,Y 616.485,Z 1097.612,A -85,B 0,C 180,E1 29262.172,E2 29262.172} C_VEL
LIN {X 0,Y 616.191,Z 1105.732,A -85,B 0,C 180,E1 29260.188,E2 29260.188} C_VEL
LIN {X 0,Y 616.026,Z 1112.678,A -85,B 0,C 180,E1 29258.118,E2 29258.118} C_VEL
LIN {X 0,Y 615.944,Z 1117.864,A -85,B 0,C 180,E1 29256.057,E2 29256.057} C_VEL
LIN {X 0,Y 615.908,Z 1121.718,A -85,B 0,C 180,E1 29253.91,E2 29253.91} C_VEL
LIN {X 0,Y 615.904,Z 1123.79,A -85,B 0,C 180,E1 29251.861,E2 29251.861} C_VEL
LIN {X 0,Y 615.896,Z 1124.425,A -85,B 0,C 180,E1 29249.628,E2 29249.628} C_VEL
LIN {X 0,Y 615.898,Z 1123.519,A -85,B 0,C 180,E1 29247.674,E2 29247.674} C_VEL
LIN {X 0,Y 615.903,Z 1120.856,A -85,B 0,C 180,E1 29245.437,E2 29245.437} C_VEL
LIN {X 0,Y 615.949,Z 1117.029,A -85,B 0,C 180,E1 29243.475,E2 29243.475} C_VEL
LIN {X 0,Y 616.055,Z 1110.899,A -85,B 0,C 180,E1 29241.224,E2 29241.224} C_VEL
LIN {X 0,Y 616.26,Z 1103.948,A -85,B 0,C 180,E1 29239.246,E2 29239.246} C_VEL
LIN {X 0,Y 616.602,Z 1094.858,A -85,B 0,C 180,E1 29237.164,E2 29237.164} C_VEL
LIN {X 0,Y 617.106,Z 1084.478,A -85,B 0,C 180,E1 29235.167,E2 29235.167} C_VEL
LIN {X 0,Y 617.774,Z 1072.594,A -85,B 0,C 180,E1 29233.256,E2 29233.256} C_VEL
LIN {X 0,Y 618.687,Z 1058.809,A -85,B 0,C 180,E1 29231.337,E2 29231.337} C_VEL
LIN {X 0,Y 619.978,Z 1041.745,A -85,B 0,C 180,E1 29229.296,E2 29229.296} C_VEL
LIN {X 0,Y 621.356,Z 1025.089,A -85,B 0,C 180,E1 29227.581,E2 29227.581} C_VEL
LIN {X 0,Y 623.033,Z 1006.145,A -85,B 0,C 180,E1 29225.893,E2 29225.893} C_VEL
LIN {X 0,Y 624.652,Z 988.004,A -85,B 0,C 180,E1 29224.495,E2 29224.495} C_VEL
LIN {X 0,Y 626.307,Z 969.037,A -85,B 0,C 180,E1 29223.243,E2 29223.243} C_VEL
LIN {X 0,Y 628.021,Z 948.789,A -85,B 0,C 180,E1 29222.09,E2 29222.09} C_VEL
LIN {X 0,Y 629.518,Z 928.47,A -85,B 0,C 180,E1 29221.128,E2 29221.128} C_VEL
LIN {X 0,Y 631.075,Z 906.409,A -85,B 0,C 180,E1 29220.258,E2 29220.258} C_VEL
LIN {X 0,Y 632.241,Z 885.575,A -85,B 0,C 180,E1 29219.607,E2 29219.607} C_VEL
LIN {X 0,Y 633.271,Z 862.99,A -85,B 0,C 180,E1 29219.057,E2 29219.057} C_VEL
LIN {X 0,Y 633.962,Z 840.613,A -85,B 0,C 180,E1 29218.68,E2 29218.68} C_VEL
LIN {X 0,Y 636.921,Z 627.7,A -85,B 0,C 180,E1 29216.055,E2 29216.055} C_VEL
LIN {X 0,Y 638.19,Z 526.123,A -85,B 0,C 180,E1 29214.792,E2 29214.792} C_VEL
LIN {X 0,Y 631.73,Z 495.574,A -85,B 0,C 180,E1 29213.9,E2 29213.9} C_VEL
LIN {X 0,Y 633.849,Z 463.382,A -85,B 0,C 180,E1 29211.412,E2 29211.412} C_VEL
LIN {X 0,Y 626.739,Z 444.593,A -85,B 0,C 180,E1 29209.268,E2 29209.268} C_VEL
LIN {X 0,Y 619.57,Z 427.068,A -85,B 0,C 180,E1 29207.112,E2 29207.112} C_VEL
LIN {X 0,Y 616.966,Z 420.545,A -85,B 0,C 180,E1 29206.238,E2 29206.238} C_VEL
LIN {X 0,Y 616.939,Z 420.383,A -85,B 0,C 180,E1 29203.575,E2 29203.575} C_VEL
LIN {X 0,Y 616.942,Z 420.351,A -85,B 0,C 180,E1 29200.291,E2 29200.291} C_VEL
LIN {X 0,Y 616.922,Z 420.373,A -85,B 0,C 180,E1 29197.664,E2 29197.664} C_VEL
LIN {X 0,Y 616.98,Z 420.352,A -85,B 0,C 180,E1 29194.557,E2 29194.557} C_VEL
LIN {X 0,Y 616.914,Z 420.374,A -85,B 0,C 180,E1 29191.678,E2 29191.678} C_VEL
LIN {X 0,Y 616.984,Z 420.371,A -85,B 0,C 180,E1 29188.747,E2 29188.747} C_VEL
LIN {X 0,Y 616.911,Z 420.38,A -85,B 0,C 180,E1 29185.688,E2 29185.688} C_VEL
LIN {X 0,Y 616.971,Z 420.379,A -85,B 0,C 180,E1 29182.757,E2 29182.757} C_VEL
LIN {X 0,Y 616.922,Z 420.379,A -85,B 0,C 180,E1 29179.665,E2 29179.665} C_VEL
LIN {X 0,Y 616.951,Z 420.369,A -85,B 0,C 180,E1 29176.864,E2 29176.864} C_VEL
LIN {X 0,Y 616.934,Z 420.374,A -85,B 0,C 180,E1 29173.688,E2 29173.688} C_VEL
LIN {X 0,Y 616.943,Z 420.376,A -85,B 0,C 180,E1 29170.931,E2 29170.931} C_VEL
LIN {X 0,Y 616.943,Z 420.37,A -85,B 0,C 180,E1 29167.637,E2 29167.637} C_VEL
LIN {X 0,Y 616.945,Z 420.378,A -85,B 0,C 180,E1 29164.928,E2 29164.928} C_VEL
LIN {X 0,Y 616.962,Z 420.376,A -85,B 0,C 180,E1 29161.672,E2 29161.672} C_VEL
LIN {X 0,Y 616.947,Z 420.363,A -85,B 0,C 180,E1 29158.886,E2 29158.886} C_VEL
LIN {X 0,Y 616.985,Z 420.367,A -85,B 0,C 180,E1 29155.725,E2 29155.725} C_VEL
LIN {X 0,Y 616.953,Z 420.375,A -85,B 0,C 180,E1 29152.831,E2 29152.831} C_VEL
LIN {X 0,Y 617.002,Z 420.364,A -85,B 0,C 180,E1 29149.731,E2 29149.731} C_VEL
LIN {X 0,Y 616.958,Z 420.375,A -85,B 0,C 180,E1 29146.79,E2 29146.79} C_VEL
LIN {X 0,Y 617.014,Z 420.37,A -85,B 0,C 180,E1 29143.719,E2 29143.719} C_VEL
LIN {X 0,Y 616.963,Z 420.369,A -85,B 0,C 180,E1 29140.694,E2 29140.694} C_VEL
LIN {X 0,Y 617.015,Z 420.363,A -85,B 0,C 180,E1 29137.515,E2 29137.515} C_VEL
LIN {X 0,Y 616.974,Z 420.369,A -85,B 0,C 180,E1 29134.463,E2 29134.463} C_VEL
LIN {X 0,Y 617.002,Z 420.363,A -85,B 0,C 180,E1 29131.229,E2 29131.229} C_VEL
LIN {X 0,Y 616.999,Z 420.364,A -85,B 0,C 180,E1 29128.109,E2 29128.109} C_VEL
LIN {X 0,Y 616.984,Z 420.351,A -85,B 0,C 180,E1 29124.878,E2 29124.878} C_VEL
LIN {X 0,Y 617.01,Z 420.345,A -85,B 0,C 180,E1 29121.753,E2 29121.753} C_VEL
LIN {X 0,Y 616.985,Z 420.376,A -85,B 0,C 180,E1 29118.608,E2 29118.608} C_VEL
LIN {X 0,Y 617.006,Z 420.338,A -85,B 0,C 180,E1 29115.483,E2 29115.483} C_VEL
LIN {X 0,Y 617.039,Z 420.721,A -85,B 0,C 180,E1 29114.469,E2 29114.469} C_VEL
LIN {X 0,Y 626.05,Z 441.995,A -85,B 0,C 180,E1 29111.883,E2 29111.883} C_VEL
LIN {X 0,Y 631.756,Z 456.209,A -85,B 0,C 180,E1 29110.32,E2 29110.32} C_VEL
LIN {X 0,Y 638.005,Z 467.213,A -85,B 0,C 180,E1 29109.708,E2 29109.708} C_VEL
LIN {X 0,Y 641.385,Z 483.916,A -85,B 0,C 180,E1 29109.236,E2 29109.236} C_VEL
LIN {X 0,Y 637.302,Z 731.643,A -85,B 0,C 180,E1 29106.056,E2 29106.056} C_VEL
LIN {X 0,Y 635.575,Z 844.147,A -85,B 0,C 180,E1 29104.62,E2 29104.62} C_VEL
LIN {X 0,Y 634.667,Z 869.618,A -85,B 0,C 180,E1 29104.136,E2 29104.136} C_VEL
LIN {X 0,Y 633.705,Z 890.306,A -85,B 0,C 180,E1 29103.613,E2 29103.613} C_VEL
LIN {X 0,Y 632.401,Z 914.511,A -85,B 0,C 180,E1 29102.842,E2 29102.842} C_VEL
LIN {X 0,Y 630.978,Z 936.319,A -85,B 0,C 180,E1 29101.986,E2 29101.986} C_VEL
LIN {X 0,Y 629.466,Z 958.948,A -85,B 0,C 180,E1 29100.932,E2 29100.932} C_VEL
LIN {X 0,Y 627.937,Z 978.787,A -85,B 0,C 180,E1 29099.842,E2 29099.842} C_VEL
LIN {X 0,Y 626.352,Z 998.683,A -85,B 0,C 180,E1 29098.597,E2 29098.597} C_VEL
LIN {X 0,Y 624.667,Z 1018.867,A -85,B 0,C 180,E1 29097.129,E2 29097.129} C_VEL
LIN {X 0,Y 623.257,Z 1035.933,A -85,B 0,C 180,E1 29095.72,E2 29095.72} C_VEL
LIN {X 0,Y 621.571,Z 1054.596,A -85,B 0,C 180,E1 29093.915,E2 29093.915} C_VEL
LIN {X 0,Y 620.303,Z 1069.621,A -85,B 0,C 180,E1 29092.26,E2 29092.26} C_VEL
LIN {X 0,Y 618.999,Z 1086.004,A -85,B 0,C 180,E1 29090.196,E2 29090.196} C_VEL
LIN {X 0,Y 618.09,Z 1098.511,A -85,B 0,C 180,E1 29088.388,E2 29088.388} C_VEL
LIN {X 0,Y 617.251,Z 1111.997,A -85,B 0,C 180,E1 29086.135,E2 29086.135} C_VEL
LIN {X 0,Y 616.755,Z 1121.557,A -85,B 0,C 180,E1 29084.266,E2 29084.266} C_VEL
LIN {X 0,Y 616.35,Z 1131.481,A -85,B 0,C 180,E1 29081.985,E2 29081.985} C_VEL
LIN {X 0,Y 616.111,Z 1138.513,A -85,B 0,C 180,E1 29080,E2 29080} C_VEL
LIN {X 0,Y 615.981,Z 1144.507,A -85,B 0,C 180,E1 29077.931,E2 29077.931} C_VEL
LIN {X 0,Y 615.92,Z 1149.405,A -85,B 0,C 180,E1 29075.642,E2 29075.642} C_VEL
LIN {X 0,Y 615.914,Z 1152.237,A -85,B 0,C 180,E1 29073.723,E2 29073.723} C_VEL
LIN {X 0,Y 615.898,Z 1154.146,A -85,B 0,C 180,E1 29071.488,E2 29071.488} C_VEL
LIN {X 0,Y 615.884,Z 1154.349,A -85,B 0,C 180,E1 29069.349,E2 29069.349} C_VEL
LIN {X 0,Y 615.892,Z 1153.359,A -85,B 0,C 180,E1 29067.395,E2 29067.395} C_VEL
LIN {X 0,Y 615.904,Z 1150.61,A -85,B 0,C 180,E1 29065.064,E2 29065.064} C_VEL
LIN {X 0,Y 615.963,Z 1146.895,A -85,B 0,C 180,E1 29063.101,E2 29063.101} C_VEL
LIN {X 0,Y 616.033,Z 1141.71,A -85,B 0,C 180,E1 29061.036,E2 29061.036} C_VEL
LIN {X 0,Y 616.228,Z 1134.307,A -85,B 0,C 180,E1 29058.772,E2 29058.772} C_VEL
LIN {X 0,Y 616.528,Z 1126.749,A -85,B 0,C 180,E1 29056.876,E2 29056.876} C_VEL
LIN {X 0,Y 617.042,Z 1116.046,A -85,B 0,C 180,E1 29054.618,E2 29054.618} C_VEL
LIN {X 0,Y 617.67,Z 1105.114,A -85,B 0,C 180,E1 29052.671,E2 29052.671} C_VEL
LIN {X 0,Y 618.547,Z 1092.117,A -85,B 0,C 180,E1 29050.647,E2 29050.647} C_VEL
LIN {X 0,Y 619.639,Z 1077.613,A -85,B 0,C 180,E1 29048.711,E2 29048.711} C_VEL
LIN {X 0,Y 620.977,Z 1061.782,A -85,B 0,C 180,E1 29046.842,E2 29046.842} C_VEL
LIN {X 0,Y 622.442,Z 1044.82,A -85,B 0,C 180,E1 29045.11,E2 29045.11} C_VEL
LIN {X 0,Y 623.662,Z 1030.821,A -85,B 0,C 180,E1 29043.839,E2 29043.839} C_VEL
LIN {X 0,Y 625.4,Z 1010.276,A -85,B 0,C 180,E1 29042.222,E2 29042.222} C_VEL
LIN {X 0,Y 626.861,Z 992.37,A -85,B 0,C 180,E1 29040.994,E2 29040.994} C_VEL
LIN {X 0,Y 628.533,Z 971.177,A -85,B 0,C 180,E1 29039.715,E2 29039.715} C_VEL
LIN {X 0,Y 630.085,Z 949.8,A -85,B 0,C 180,E1 29038.623,E2 29038.623} C_VEL
LIN {X 0,Y 631.614,Z 927.659,A -85,B 0,C 180,E1 29037.651,E2 29037.651} C_VEL
LIN {X 0,Y 632.961,Z 904.29,A -85,B 0,C 180,E1 29036.813,E2 29036.813} C_VEL
LIN {X 0,Y 634.074,Z 882.622,A -85,B 0,C 180,E1 29036.175,E2 29036.175} C_VEL
LIN {X 0,Y 635.11,Z 857.602,A -85,B 0,C 180,E1 29035.615,E2 29035.615} C_VEL
LIN {X 0,Y 635.771,Z 835.456,A -85,B 0,C 180,E1 29035.256,E2 29035.256} C_VEL
LIN {X 0,Y 639.448,Z 594.351,A -85,B 0,C 180,E1 29032.19,E2 29032.19} C_VEL
LIN {X 0,Y 641.247,Z 482.314,A -85,B 0,C 180,E1 29030.732,E2 29030.732} C_VEL
LIN {X 0,Y 637.513,Z 465.919,A -85,B 0,C 180,E1 29030.24,E2 29030.24} C_VEL
LIN {X 0,Y 631.478,Z 455.621,A -85,B 0,C 180,E1 29029.638,E2 29029.638} C_VEL
LIN {X 0,Y 623.129,Z 435.015,A -85,B 0,C 180,E1 29027.301,E2 29027.301} C_VEL
LIN {X 0,Y 617.039,Z 420.724,A -85,B 0,C 180,E1 29025.531,E2 29025.531} C_VEL
LIN {X 0,Y 617.005,Z 420.341,A -85,B 0,C 180,E1 29024.694,E2 29024.694} C_VEL
LIN {X 0,Y 616.984,Z 420.377,A -85,B 0,C 180,E1 29021.516,E2 29021.516} C_VEL
LIN {X 0,Y 617.007,Z 420.343,A -85,B 0,C 180,E1 29018.365,E2 29018.365} C_VEL
LIN {X 0,Y 616.977,Z 420.359,A -85,B 0,C 180,E1 29015.35,E2 29015.35} C_VEL
LIN {X 0,Y 617.012,Z 420.355,A -85,B 0,C 180,E1 29012.219,E2 29012.219} C_VEL
LIN {X 0,Y 616.977,Z 420.365,A -85,B 0,C 180,E1 29009.129,E2 29009.129} C_VEL
LIN {X 0,Y 617.009,Z 420.364,A -85,B 0,C 180,E1 29005.948,E2 29005.948} C_VEL
LIN {X 0,Y 616.978,Z 420.368,A -85,B 0,C 180,E1 29002.889,E2 29002.889} C_VEL
LIN {X 0,Y 616.984,Z 420.371,A -85,B 0,C 180,E1 28999.601,E2 28999.601} C_VEL
LIN {X 0,Y 616.99,Z 420.37,A -85,B 0,C 180,E1 28996.572,E2 28996.572} C_VEL
LIN {X 0,Y 616.968,Z 420.372,A -85,B 0,C 180,E1 28993.4,E2 28993.4} C_VEL
LIN {X 0,Y 616.985,Z 420.368,A -85,B 0,C 180,E1 28990.458,E2 28990.458} C_VEL
LIN {X 0,Y 616.962,Z 420.376,A -85,B 0,C 180,E1 28987.262,E2 28987.262} C_VEL
LIN {X 0,Y 616.977,Z 420.366,A -85,B 0,C 180,E1 28984.368,E2 28984.368} C_VEL
LIN {X 0,Y 616.957,Z 420.363,A -85,B 0,C 180,E1 28981.207,E2 28981.207} C_VEL
LIN {X 0,Y 616.958,Z 420.376,A -85,B 0,C 180,E1 28978.421,E2 28978.421} C_VEL
LIN {X 0,Y 616.958,Z 420.377,A -85,B 0,C 180,E1 28975.166,E2 28975.166} C_VEL
LIN {X 0,Y 616.942,Z 420.37,A -85,B 0,C 180,E1 28972.456,E2 28972.456} C_VEL
LIN {X 0,Y 616.972,Z 420.376,A -85,B 0,C 180,E1 28969.259,E2 28969.259} C_VEL
LIN {X 0,Y 616.934,Z 420.374,A -85,B 0,C 180,E1 28966.408,E2 28966.408} C_VEL
LIN {X 0,Y 616.987,Z 420.364,A -85,B 0,C 180,E1 28963.331,E2 28963.331} C_VEL
LIN {X 0,Y 616.926,Z 420.378,A -85,B 0,C 180,E1 28960.397,E2 28960.397} C_VEL
LIN {X 0,Y 616.994,Z 420.379,A -85,B 0,C 180,E1 28957.313,E2 28957.313} C_VEL
LIN {X 0,Y 616.919,Z 420.378,A -85,B 0,C 180,E1 28954.358,E2 28954.358} C_VEL
LIN {X 0,Y 616.998,Z 420.367,A -85,B 0,C 180,E1 28951.335,E2 28951.335} C_VEL
LIN {X 0,Y 616.912,Z 420.373,A -85,B 0,C 180,E1 28948.431,E2 28948.431} C_VEL
LIN {X 0,Y 616.95,Z 420.362,A -85,B 0,C 180,E1 28945.583,E2 28945.583} C_VEL
LIN {X 0,Y 616.917,Z 420.367,A -85,B 0,C 180,E1 28942.426,E2 28942.426} C_VEL
LIN {X 0,Y 616.922,Z 420.359,A -85,B 0,C 180,E1 28939.829,E2 28939.829} C_VEL
LIN {X 0,Y 616.945,Z 420.385,A -85,B 0,C 180,E1 28936.592,E2 28936.592} C_VEL
LIN {X 0,Y 616.933,Z 420.406,A -85,B 0,C 180,E1 28933.794,E2 28933.794} C_VEL
LIN {X 0,Y 617.044,Z 420.979,A -85,B 0,C 180,E1 28933.586,E2 28933.586} C_VEL
LIN {X 0,Y 625.486,Z 441.428,A -85,B 0,C 180,E1 28931.015,E2 28931.015} C_VEL
LIN {X 0,Y 632.901,Z 460.936,A -85,B 0,C 180,E1 28928.77,E2 28928.77} C_VEL
LIN {X 0,Y 633.821,Z 463.728,A -85,B 0,C 180,E1 28928.469,E2 28928.469} C_VEL
LIN {X 0,Y 633.388,Z 470.059,A -85,B 0,C 180,E1 28927.974,E2 28927.974} C_VEL
LIN {X 0,Y 632.251,Z 474.243,A -85,B 0,C 180,E1 28927.71,E2 28927.71} C_VEL
LIN {X 0,Y 626.172,Z 485.972,A -85,B 0,C 180,E1 28927.171,E2 28927.171} C_VEL
LIN {X 0,Y 625.272,Z 489.564,A -85,B 0,C 180,E1 28926.938,E2 28926.938} C_VEL
LIN {X 0,Y 625.011,Z 496.288,A -85,B 0,C 180,E1 28926.45,E2 28926.45} C_VEL
LIN {X 0,Y 631.952,Z 529.018,A -85,B 0,C 180,E1 28925.507,E2 28925.507} C_VEL
LIN {X 0,Y 628.127,Z 795.021,A -85,B 0,C 180,E1 28922.219,E2 28922.219} C_VEL
LIN {X 0,Y 627.202,Z 849.422,A -85,B 0,C 180,E1 28921.521,E2 28921.521} C_VEL
LIN {X 0,Y 626.295,Z 871.781,A -85,B 0,C 180,E1 28921.073,E2 28921.073} C_VEL
LIN {X 0,Y 625.179,Z 893.484,A -85,B 0,C 180,E1 28920.494,E2 28920.494} C_VEL
LIN {X 0,Y 623.731,Z 914.95,A -85,B 0,C 180,E1 28919.746,E2 28919.746} C_VEL
LIN {X 0,Y 622.122,Z 936.56,A -85,B 0,C 180,E1 28918.827,E2 28918.827} C_VEL
LIN {X 0,Y 620.443,Z 956.101,A -85,B 0,C 180,E1 28917.817,E2 28917.817} C_VEL
LIN {X 0,Y 618.611,Z 976.3,A -85,B 0,C 180,E1 28916.598,E2 28916.598} C_VEL
LIN {X 0,Y 616.911,Z 994.15,A -85,B 0,C 180,E1 28915.334,E2 28915.334} C_VEL
LIN {X 0,Y 615.036,Z 1013.487,A -85,B 0,C 180,E1 28913.752,E2 28913.752} C_VEL
LIN {X 0,Y 613.521,Z 1029.711,A -85,B 0,C 180,E1 28912.216,E2 28912.216} C_VEL
LIN {X 0,Y 612.054,Z 1045.808,A -85,B 0,C 180,E1 28910.463,E2 28910.463} C_VEL
LIN {X 0,Y 610.838,Z 1060.607,A -85,B 0,C 180,E1 28908.615,E2 28908.615} C_VEL
LIN {X 0,Y 609.723,Z 1075.817,A -85,B 0,C 180,E1 28906.384,E2 28906.384} C_VEL
LIN {X 0,Y 609.019,Z 1087.607,A -85,B 0,C 180,E1 28904.354,E2 28904.354} C_VEL
LIN {X 0,Y 608.539,Z 1097.615,A -85,B 0,C 180,E1 28902.334,E2 28902.334} C_VEL
LIN {X 0,Y 608.223,Z 1105.734,A -85,B 0,C 180,E1 28900.323,E2 28900.323} C_VEL
LIN {X 0,Y 608.044,Z 1112.68,A -85,B 0,C 180,E1 28898.225,E2 28898.225} C_VEL
LIN {X 0,Y 607.952,Z 1117.865,A -85,B 0,C 180,E1 28896.137,E2 28896.137} C_VEL
LIN {X 0,Y 607.91,Z 1121.718,A -85,B 0,C 180,E1 28893.961,E2 28893.961} C_VEL
LIN {X 0,Y 607.906,Z 1123.789,A -85,B 0,C 180,E1 28891.885,E2 28891.885} C_VEL
LIN {X 0,Y 607.896,Z 1124.425,A -85,B 0,C 180,E1 28889.623,E2 28889.623} C_VEL
LIN {X 0,Y 607.898,Z 1123.518,A -85,B 0,C 180,E1 28887.643,E2 28887.643} C_VEL
LIN {X 0,Y 607.904,Z 1120.855,A -85,B 0,C 180,E1 28885.377,E2 28885.377} C_VEL
LIN {X 0,Y 607.95,Z 1117.028,A -85,B 0,C 180,E1 28883.389,E2 28883.389} C_VEL
LIN {X 0,Y 608.068,Z 1110.897,A -85,B 0,C 180,E1 28881.108,E2 28881.108} C_VEL
LIN {X 0,Y 608.289,Z 1103.946,A -85,B 0,C 180,E1 28879.104,E2 28879.104} C_VEL
LIN {X 0,Y 608.664,Z 1094.854,A -85,B 0,C 180,E1 28876.994,E2 28876.994} C_VEL
LIN {X 0,Y 609.21,Z 1084.476,A -85,B 0,C 180,E1 28874.97,E2 28874.97} C_VEL
LIN {X 0,Y 609.977,Z 1072.005,A -85,B 0,C 180,E1 28872.937,E2 28872.937} C_VEL
LIN {X 0,Y 611.124,Z 1056.78,A -85,B 0,C 180,E1 28870.8,E2 28870.8} C_VEL
LIN {X 0,Y 612.371,Z 1042.414,A -85,B 0,C 180,E1 28869.048,E2 28869.048} C_VEL
LIN {X 0,Y 613.811,Z 1026.297,A -85,B 0,C 180,E1 28867.356,E2 28867.356} C_VEL
LIN {X 0,Y 615.529,Z 1008.626,A -85,B 0,C 180,E1 28865.733,E2 28865.733} C_VEL
LIN {X 0,Y 617.224,Z 990.746,A -85,B 0,C 180,E1 28864.32,E2 28864.32} C_VEL
LIN {X 0,Y 619.195,Z 969.965,A -85,B 0,C 180,E1 28862.91,E2 28862.91} C_VEL
LIN {X 0,Y 620.932,Z 950.719,A -85,B 0,C 180,E1 28861.795,E2 28861.795} C_VEL
LIN {X 0,Y 622.619,Z 929.782,A -85,B 0,C 180,E1 28860.777,E2 28860.777} C_VEL
LIN {X 0,Y 624.251,Z 908.311,A -85,B 0,C 180,E1 28859.911,E2 28859.911} C_VEL
LIN {X 0,Y 625.547,Z 886.497,A -85,B 0,C 180,E1 28859.216,E2 28859.216} C_VEL
LIN {X 0,Y 626.644,Z 864.22,A -85,B 0,C 180,E1 28858.663,E2 28858.663} C_VEL
LIN {X 0,Y 627.377,Z 841.42,A -85,B 0,C 180,E1 28858.273,E2 28858.273} C_VEL
LIN {X 0,Y 630.566,Z 619.419,A -85,B 0,C 180,E1 28855.525,E2 28855.525} C_VEL
LIN {X 0,Y 631.801,Z 527.779,A -85,B 0,C 180,E1 28854.375,E2 28854.375} C_VEL
LIN {X 0,Y 624.926,Z 495.358,A -85,B 0,C 180,E1 28853.415,E2 28853.415} C_VEL
LIN {X 0,Y 626.895,Z 466.773,A -85,B 0,C 180,E1 28851.183,E2 28851.183} C_VEL
LIN {X 0,Y 619.845,Z 448.109,A -85,B 0,C 180,E1 28849.021,E2 28849.021} C_VEL
LIN {X 0,Y 612.739,Z 430.636,A -85,B 0,C 180,E1 28846.839,E2 28846.839} C_VEL
LIN {X 0,Y 609.028,Z 421.548,A -85,B 0,C 180,E1 28845.612,E2 28845.612} C_VEL
LIN {X 0,Y 609.049,Z 421.349,A -85,B 0,C 180,E1 28842.69,E2 28842.69} C_VEL
LIN {X 0,Y 608.983,Z 421.353,A -85,B 0,C 180,E1 28839.788,E2 28839.788} C_VEL
LIN {X 0,Y 609.055,Z 421.325,A -85,B 0,C 180,E1 28836.815,E2 28836.815} C_VEL
LIN {X 0,Y 608.979,Z 421.37,A -85,B 0,C 180,E1 28833.709,E2 28833.709} C_VEL
LIN {X 0,Y 609.06,Z 421.358,A -85,B 0,C 180,E1 28830.655,E2 28830.655} C_VEL
LIN {X 0,Y 608.972,Z 421.365,A -85,B 0,C 180,E1 28827.583,E2 28827.583} C_VEL
LIN {X 0,Y 609.052,Z 421.354,A -85,B 0,C 180,E1 28824.542,E2 28824.542} C_VEL
LIN {X 0,Y 608.975,Z 421.365,A -85,B 0,C 180,E1 28821.58,E2 28821.58} C_VEL
LIN {X 0,Y 609.054,Z 421.367,A -85,B 0,C 180,E1 28818.572,E2 28818.572} C_VEL
LIN {X 0,Y 608.985,Z 421.367,A -85,B 0,C 180,E1 28815.464,E2 28815.464} C_VEL
LIN {X 0,Y 609.04,Z 421.353,A -85,B 0,C 180,E1 28812.612,E2 28812.612} C_VEL
LIN {X 0,Y 608.996,Z 421.364,A -85,B 0,C 180,E1 28809.545,E2 28809.545} C_VEL
LIN {X 0,Y 609.025,Z 421.361,A -85,B 0,C 180,E1 28806.694,E2 28806.694} C_VEL
LIN {X 0,Y 609.004,Z 421.353,A -85,B 0,C 180,E1 28803.483,E2 28803.483} C_VEL
LIN {X 0,Y 609.027,Z 421.368,A -85,B 0,C 180,E1 28800.658,E2 28800.658} C_VEL
LIN {X 0,Y 609.018,Z 421.365,A -85,B 0,C 180,E1 28797.459,E2 28797.459} C_VEL
LIN {X 0,Y 609.035,Z 421.353,A -85,B 0,C 180,E1 28794.536,E2 28794.536} C_VEL
LIN {X 0,Y 609.021,Z 421.36,A -85,B 0,C 180,E1 28791.312,E2 28791.312} C_VEL
LIN {X 0,Y 609.05,Z 421.363,A -85,B 0,C 180,E1 28788.35,E2 28788.35} C_VEL
LIN {X 0,Y 609.024,Z 421.356,A -85,B 0,C 180,E1 28785.16,E2 28785.16} C_VEL
LIN {X 0,Y 609.067,Z 421.351,A -85,B 0,C 180,E1 28782.122,E2 28782.122} C_VEL
LIN {X 0,Y 609.027,Z 421.362,A -85,B 0,C 180,E1 28778.927,E2 28778.927} C_VEL
LIN {X 0,Y 609.078,Z 421.362,A -85,B 0,C 180,E1 28775.872,E2 28775.872} C_VEL
LIN {X 0,Y 609.032,Z 421.364,A -85,B 0,C 180,E1 28772.738,E2 28772.738} C_VEL
LIN {X 0,Y 609.077,Z 421.364,A -85,B 0,C 180,E1 28769.627,E2 28769.627} C_VEL
LIN {X 0,Y 609.033,Z 421.324,A -85,B 0,C 180,E1 28766.514,E2 28766.514} C_VEL
LIN {X 0,Y 609.076,Z 421.363,A -85,B 0,C 180,E1 28763.304,E2 28763.304} C_VEL
LIN {X 0,Y 609.053,Z 421.324,A -85,B 0,C 180,E1 28760.065,E2 28760.065} C_VEL
LIN {X 0,Y 609.055,Z 421.328,A -85,B 0,C 180,E1 28756.796,E2 28756.796} C_VEL
LIN {X 0,Y 609.105,Z 421.585,A -85,B 0,C 180,E1 28755.134,E2 28755.134} C_VEL
LIN {X 0,Y 612.126,Z 428.816,A -85,B 0,C 180,E1 28754.185,E2 28754.185} C_VEL
LIN {X 0,Y 620.757,Z 449.334,A -85,B 0,C 180,E1 28751.701,E2 28751.701} C_VEL
LIN {X 0,Y 623.742,Z 456.654,A -85,B 0,C 180,E1 28750.901,E2 28750.901} C_VEL
LIN {X 0,Y 632.128,Z 471.134,A -85,B 0,C 180,E1 28750.066,E2 28750.066} C_VEL
LIN {X 0,Y 634.998,Z 485.58,A -85,B 0,C 180,E1 28749.654,E2 28749.654} C_VEL
LIN {X 0,Y 630.533,Z 736.337,A -85,B 0,C 180,E1 28746.394,E2 28746.394} C_VEL
LIN {X 0,Y 628.722,Z 844.275,A -85,B 0,C 180,E1 28744.996,E2 28744.996} C_VEL
LIN {X 0,Y 627.771,Z 869.446,A -85,B 0,C 180,E1 28744.512,E2 28744.512} C_VEL
LIN {X 0,Y 626.763,Z 889.911,A -85,B 0,C 180,E1 28743.991,E2 28743.991} C_VEL
LIN {X 0,Y 625.37,Z 914.403,A -85,B 0,C 180,E1 28743.204,E2 28743.204} C_VEL
LIN {X 0,Y 623.897,Z 935.668,A -85,B 0,C 180,E1 28742.364,E2 28742.364} C_VEL
LIN {X 0,Y 622.312,Z 958.056,A -85,B 0,C 180,E1 28741.317,E2 28741.317} C_VEL
LIN {X 0,Y 620.641,Z 978.644,A -85,B 0,C 180,E1 28740.176,E2 28740.176} C_VEL
LIN {X 0,Y 618.988,Z 998.289,A -85,B 0,C 180,E1 28738.934,E2 28738.934} C_VEL
LIN {X 0,Y 617.184,Z 1018.567,A -85,B 0,C 180,E1 28737.446,E2 28737.446} C_VEL
LIN {X 0,Y 615.682,Z 1035.822,A -85,B 0,C 180,E1 28736.008,E2 28736.008} C_VEL
LIN {X 0,Y 614.007,Z 1054.532,A -85,B 0,C 180,E1 28734.224,E2 28734.224} C_VEL
LIN {X 0,Y 612.849,Z 1067.451,A -85,B 0,C 180,E1 28732.805,E2 28732.805} C_VEL
LIN {X 0,Y 611.524,Z 1082.996,A -85,B 0,C 180,E1 28730.882,E2 28730.882} C_VEL
LIN {X 0,Y 610.382,Z 1097.239,A -85,B 0,C 180,E1 28728.827,E2 28728.827} C_VEL
LIN {X 0,Y 609.534,Z 1109.688,A -85,B 0,C 180,E1 28726.781,E2 28726.781} C_VEL
LIN {X 0,Y 608.884,Z 1120.639,A -85,B 0,C 180,E1 28724.649,E2 28724.649} C_VEL
LIN {X 0,Y 608.448,Z 1129.988,A -85,B 0,C 180,E1 28722.528,E2 28722.528} C_VEL
LIN {X 0,Y 608.157,Z 1137.907,A -85,B 0,C 180,E1 28720.324,E2 28720.324} C_VEL
LIN {X 0,Y 608.026,Z 1143.745,A -85,B 0,C 180,E1 28718.321,E2 28718.321} C_VEL
LIN {X 0,Y 607.944,Z 1149.015,A -85,B 0,C 180,E1 28715.948,E2 28715.948} C_VEL
LIN {X 0,Y 607.916,Z 1152.123,A -85,B 0,C 180,E1 28713.867,E2 28713.867} C_VEL
LIN {X 0,Y 607.898,Z 1154.103,A -85,B 0,C 180,E1 28711.602,E2 28711.602} C_VEL
LIN {X 0,Y 607.884,Z 1154.372,A -85,B 0,C 180,E1 28709.435,E2 28709.435} C_VEL
LIN {X 0,Y 607.895,Z 1153.427,A -85,B 0,C 180,E1 28707.455,E2 28707.455} C_VEL
LIN {X 0,Y 607.911,Z 1150.928,A -85,B 0,C 180,E1 28705.188,E2 28705.188} C_VEL
LIN {X 0,Y 607.964,Z 1147.102,A -85,B 0,C 180,E1 28703.104,E2 28703.104} C_VEL
LIN {X 0,Y 608.033,Z 1142.219,A -85,B 0,C 180,E1 28701.108,E2 28701.108} C_VEL
LIN {X 0,Y 608.248,Z 1134.66,A -85,B 0,C 180,E1 28698.719,E2 28698.719} C_VEL
LIN {X 0,Y 608.58,Z 1126.748,A -85,B 0,C 180,E1 28696.702,E2 28696.702} C_VEL
LIN {X 0,Y 609.122,Z 1116.402,A -85,B 0,C 180,E1 28694.48,E2 28694.48} C_VEL
LIN {X 0,Y 609.829,Z 1105.112,A -85,B 0,C 180,E1 28692.441,E2 28692.441} C_VEL
LIN {X 0,Y 610.777,Z 1092.116,A -85,B 0,C 180,E1 28690.391,E2 28690.391} C_VEL
LIN {X 0,Y 611.884,Z 1078.381,A -85,B 0,C 180,E1 28688.528,E2 28688.528} C_VEL
LIN {X 0,Y 613.286,Z 1062.857,A -85,B 0,C 180,E1 28686.66,E2 28686.66} C_VEL
LIN {X 0,Y 614.744,Z 1046.234,A -85,B 0,C 180,E1 28684.955,E2 28684.955} C_VEL
LIN {X 0,Y 616.215,Z 1029.546,A -85,B 0,C 180,E1 28683.446,E2 28683.446} C_VEL
LIN {X 0,Y 618.068,Z 1008.763,A -85,B 0,C 180,E1 28681.81,E2 28681.81} C_VEL
LIN {X 0,Y 619.623,Z 990.714,A -85,B 0,C 180,E1 28680.569,E2 28680.569} C_VEL
LIN {X 0,Y 621.554,Z 967.33,A -85,B 0,C 180,E1 28679.178,E2 28679.178} C_VEL
LIN {X 0,Y 623.068,Z 947.795,A -85,B 0,C 180,E1 28678.185,E2 28678.185} C_VEL
LIN {X 0,Y 624.723,Z 924.362,A -85,B 0,C 180,E1 28677.17,E2 28677.17} C_VEL
LIN {X 0,Y 626.035,Z 902.681,A -85,B 0,C 180,E1 28676.398,E2 28676.398} C_VEL
LIN {X 0,Y 627.336,Z 878.61,A -85,B 0,C 180,E1 28675.699,E2 28675.699} C_VEL
LIN {X 0,Y 628.34,Z 855.33,A -85,B 0,C 180,E1 28675.198,E2 28675.198} C_VEL
LIN {X 0,Y 629.063,Z 830.589,A -85,B 0,C 180,E1 28674.807,E2 28674.807} C_VEL
LIN {X 0,Y 632.946,Z 595.108,A -85,B 0,C 180,E1 28671.776,E2 28671.776} C_VEL
LIN {X 0,Y 634.829,Z 483.874,A -85,B 0,C 180,E1 28670.31,E2 28670.31} C_VEL
LIN {X 0,Y 631.734,Z 470.15,A -85,B 0,C 180,E1 28669.893,E2 28669.893} C_VEL
LIN {X 0,Y 623.466,Z 456.076,A -85,B 0,C 180,E1 28669.058,E2 28669.058} C_VEL
LIN {X 0,Y 615.136,Z 435.793,A -85,B 0,C 180,E1 28666.689,E2 28666.689} C_VEL
LIN {X 0,Y 609.128,Z 421.714,A -85,B 0,C 180,E1 28664.899,E2 28664.899} C_VEL
LIN {X 0,Y 609.067,Z 421.322,A -85,B 0,C 180,E1 28664.244,E2 28664.244} C_VEL
LIN {X 0,Y 609.072,Z 421.348,A -85,B 0,C 180,E1 28660.96,E2 28660.96} C_VEL
LIN {X 0,Y 609.048,Z 421.348,A -85,B 0,C 180,E1 28657.761,E2 28657.761} C_VEL
LIN {X 0,Y 609.07,Z 421.323,A -85,B 0,C 180,E1 28654.612,E2 28654.612} C_VEL
LIN {X 0,Y 609.039,Z 421.367,A -85,B 0,C 180,E1 28651.472,E2 28651.472} C_VEL
LIN {X 0,Y 609.08,Z 421.353,A -85,B 0,C 180,E1 28648.367,E2 28648.367} C_VEL
LIN {X 0,Y 609.033,Z 421.36,A -85,B 0,C 180,E1 28645.228,E2 28645.228} C_VEL
LIN {X 0,Y 609.077,Z 421.349,A -85,B 0,C 180,E1 28642.082,E2 28642.082} C_VEL
LIN {X 0,Y 609.029,Z 421.355,A -85,B 0,C 180,E1 28638.97,E2 28638.97} C_VEL
LIN {X 0,Y 609.059,Z 421.361,A -85,B 0,C 180,E1 28635.717,E2 28635.717} C_VEL
LIN {X 0,Y 609.029,Z 421.361,A -85,B 0,C 180,E1 28632.709,E2 28632.709} C_VEL
LIN {X 0,Y 609.036,Z 421.355,A -85,B 0,C 180,E1 28629.449,E2 28629.449} C_VEL
LIN {X 0,Y 609.032,Z 421.361,A -85,B 0,C 180,E1 28626.505,E2 28626.505} C_VEL
LIN {X 0,Y 609.021,Z 421.367,A -85,B 0,C 180,E1 28623.2,E2 28623.2} C_VEL
LIN {X 0,Y 609.034,Z 421.349,A -85,B 0,C 180,E1 28620.282,E2 28620.282} C_VEL
LIN {X 0,Y 609.011,Z 421.355,A -85,B 0,C 180,E1 28617.083,E2 28617.083} C_VEL
LIN {X 0,Y 609.032,Z 421.363,A -85,B 0,C 180,E1 28614.158,E2 28614.158} C_VEL
LIN {X 0,Y 609.003,Z 421.365,A -85,B 0,C 180,E1 28610.931,E2 28610.931} C_VEL
LIN {X 0,Y 609.024,Z 421.36,A -85,B 0,C 180,E1 28608.061,E2 28608.061} C_VEL
LIN {X 0,Y 608.999,Z 421.367,A -85,B 0,C 180,E1 28604.867,E2 28604.867} C_VEL
LIN {X 0,Y 609.011,Z 421.361,A -85,B 0,C 180,E1 28602.021,E2 28602.021} C_VEL
LIN {X 0,Y 608.995,Z 421.361,A -85,B 0,C 180,E1 28598.825,E2 28598.825} C_VEL
LIN {X 0,Y 608.989,Z 421.366,A -85,B 0,C 180,E1 28596.14,E2 28596.14} C_VEL
LIN {X 0,Y 609.01,Z 421.365,A -85,B 0,C 180,E1 28592.949,E2 28592.949} C_VEL
LIN {X 0,Y 608.978,Z 421.371,A -85,B 0,C 180,E1 28590.165,E2 28590.165} C_VEL
LIN {X 0,Y 609.033,Z 421.371,A -85,B 0,C 180,E1 28587.083,E2 28587.083} C_VEL
LIN {X 0,Y 608.969,Z 421.328,A -85,B 0,C 180,E1 28584.114,E2 28584.114} C_VEL
LIN {X 0,Y 609.047,Z 421.365,A -85,B 0,C 180,E1 28581.039,E2 28581.039} C_VEL
LIN {X 0,Y 608.976,Z 421.337,A -85,B 0,C 180,E1 28578.056,E2 28578.056} C_VEL
LIN {X 0,Y 609.056,Z 421.328,A -85,B 0,C 180,E1 28575.038,E2 28575.038} C_VEL
LIN {X 0,Y 609.037,Z 421.677,A -85,B 0,C 180,E1 28574.26,E2 28574.26} C_VEL
LIN {X 0,Y 615.52,Z 437.403,A -85,B 0,C 180,E1 28572.204,E2 28572.204} C_VEL
LIN {X 0,Y 622.923,Z 456.044,A -85,B 0,C 180,E1 28569.946,E2 28569.946} C_VEL
LIN {X 0,Y 626.896,Z 467.066,A -85,B 0,C 180,E1 28568.7,E2 28568.7} C_VEL
LIN {X 0,Y 625.272,Z 489.564,A -85,B 0,C 180,E1 28566.938,E2 28566.938} C_VEL
LIN {X 0,Y 624.949,Z 494.201,A -85,B 0,C 180,E1 28566.669,E2 28566.669} C_VEL
LIN {X 0,Y 624.42,Z 501.572,A -85,B 0,C 180,E1 28566.451,E2 28566.451} C_VEL
LIN {X 0,Y 623.738,Z 518.429,A -85,B 0,C 180,E1 28566.235,E2 28566.235} C_VEL
LIN {X 0,Y 624.328,Z 523.905,A -85,B 0,C 180,E1 28566.115,E2 28566.115} C_VEL
LIN {X 0,Y 625.569,Z 531.212,A -85,B 0,C 180,E1 28565.925,E2 28565.925} C_VEL
LIN {X 0,Y 621.506,Z 799.563,A -85,B 0,C 180,E1 28562.585,E2 28562.585} C_VEL
LIN {X 0,Y 620.611,Z 850.14,A -85,B 0,C 180,E1 28561.932,E2 28561.932} C_VEL
LIN {X 0,Y 619.671,Z 872.324,A -85,B 0,C 180,E1 28561.483,E2 28561.483} C_VEL
LIN {X 0,Y 618.527,Z 893.763,A -85,B 0,C 180,E1 28560.908,E2 28560.908} C_VEL
LIN {X 0,Y 617.007,Z 915.199,A -85,B 0,C 180,E1 28560.157,E2 28560.157} C_VEL
LIN {X 0,Y 615.303,Z 936.788,A -85,B 0,C 180,E1 28559.232,E2 28559.232} C_VEL
LIN {X 0,Y 613.512,Z 956.46,A -85,B 0,C 180,E1 28558.206,E2 28558.206} C_VEL
LIN {X 0,Y 611.585,Z 976.303,A -85,B 0,C 180,E1 28556.997,E2 28556.997} C_VEL
LIN {X 0,Y 609.73,Z 994.316,A -85,B 0,C 180,E1 28555.706,E2 28555.706} C_VEL
LIN {X 0,Y 607.699,Z 1013.91,A -85,B 0,C 180,E1 28554.083,E2 28554.083} C_VEL
LIN {X 0,Y 606.039,Z 1030.34,A -85,B 0,C 180,E1 28552.506,E2 28552.506} C_VEL
LIN {X 0,Y 604.45,Z 1046.309,A -85,B 0,C 180,E1 28550.732,E2 28550.732} C_VEL
LIN {X 0,Y 603.137,Z 1061.045,A -85,B 0,C 180,E1 28548.861,E2 28548.861} C_VEL
LIN {X 0,Y 602.049,Z 1074.238,A -85,B 0,C 180,E1 28546.896,E2 28546.896} C_VEL
LIN {X 0,Y 601.158,Z 1087.175,A -85,B 0,C 180,E1 28544.644,E2 28544.644} C_VEL
LIN {X 0,Y 600.575,Z 1098.025,A -85,B 0,C 180,E1 28542.402,E2 28542.402} C_VEL
LIN {X 0,Y 600.242,Z 1106.089,A -85,B 0,C 180,E1 28540.364,E2 28540.364} C_VEL
LIN {X 0,Y 600.037,Z 1113.19,A -85,B 0,C 180,E1 28538.143,E2 28538.143} C_VEL
LIN {X 0,Y 599.952,Z 1118.073,A -85,B 0,C 180,E1 28536.123,E2 28536.123} C_VEL
LIN {X 0,Y 599.904,Z 1121.946,A -85,B 0,C 180,E1 28533.823,E2 28533.823} C_VEL
LIN {X 0,Y 599.902,Z 1123.857,A -85,B 0,C 180,E1 28531.815,E2 28531.815} C_VEL
LIN {X 0,Y 599.894,Z 1124.402,A -85,B 0,C 180,E1 28529.522,E2 28529.522} C_VEL
LIN {X 0,Y 599.895,Z 1123.449,A -85,B 0,C 180,E1 28527.516,E2 28527.516} C_VEL
LIN {X 0,Y 599.906,Z 1120.694,A -85,B 0,C 180,E1 28525.22,E2 28525.22} C_VEL
LIN {X 0,Y 599.955,Z 1116.82,A -85,B 0,C 180,E1 28523.204,E2 28523.204} C_VEL
LIN {X 0,Y 600.085,Z 1110.895,A -85,B 0,C 180,E1 28520.989,E2 28520.989} C_VEL
LIN {X 0,Y 600.321,Z 1103.943,A -85,B 0,C 180,E1 28518.957,E2 28518.957} C_VEL
LIN {X 0,Y 600.73,Z 1094.851,A -85,B 0,C 180,E1 28516.819,E2 28516.819} C_VEL
LIN {X 0,Y 601.374,Z 1083.94,A -85,B 0,C 180,E1 28514.657,E2 28514.657} C_VEL
LIN {X 0,Y 602.192,Z 1072.227,A -85,B 0,C 180,E1 28512.697,E2 28512.697} C_VEL
LIN {X 0,Y 603.384,Z 1057.985,A -85,B 0,C 180,E1 28510.644,E2 28510.644} C_VEL
LIN {X 0,Y 604.742,Z 1043.425,A -85,B 0,C 180,E1 28508.833,E2 28508.833} C_VEL
LIN {X 0,Y 606.318,Z 1027.258,A -85,B 0,C 180,E1 28507.096,E2 28507.096} C_VEL
LIN {X 0,Y 608.144,Z 1009.947,A -85,B 0,C 180,E1 28505.471,E2 28505.471} C_VEL
LIN {X 0,Y 610.006,Z 991.555,A -85,B 0,C 180,E1 28503.993,E2 28503.993} C_VEL
LIN {X 0,Y 612.118,Z 970.968,A -85,B 0,C 180,E1 28502.571,E2 28502.571} C_VEL
LIN {X 0,Y 613.868,Z 952.7,A -85,B 0,C 180,E1 28501.494,E2 28501.494} C_VEL
LIN {X 0,Y 615.746,Z 931.109,A -85,B 0,C 180,E1 28500.419,E2 28500.419} C_VEL
LIN {X 0,Y 617.343,Z 911.027,A -85,B 0,C 180,E1 28499.592,E2 28499.592} C_VEL
LIN {X 0,Y 618.815,Z 888.401,A -85,B 0,C 180,E1 28498.848,E2 28498.848} C_VEL
LIN {X 0,Y 619.894,Z 867.752,A -85,B 0,C 180,E1 28498.319,E2 28498.319} C_VEL
LIN {X 0,Y 620.737,Z 844.055,A -85,B 0,C 180,E1 28497.888,E2 28497.888} C_VEL
LIN {X 0,Y 624.103,Z 621.288,A -85,B 0,C 180,E1 28495.111,E2 28495.111} C_VEL
LIN {X 0,Y 625.414,Z 529.249,A -85,B 0,C 180,E1 28493.945,E2 28493.945} C_VEL
LIN {X 0,Y 618.157,Z 495.185,A -85,B 0,C 180,E1 28492.922,E2 28492.922} C_VEL
LIN {X 0,Y 619.968,Z 470.224,A -85,B 0,C 180,E1 28490.955,E2 28490.955} C_VEL
LIN {X 0,Y 613.312,Z 452.436,A -85,B 0,C 180,E1 28488.869,E2 28488.869} C_VEL
LIN {X 0,Y 605.857,Z 433.758,A -85,B 0,C 180,E1 28486.511,E2 28486.511} C_VEL
LIN {X 0,Y 601.165,Z 422.622,A -85,B 0,C 180,E1 28484.982,E2 28484.982} C_VEL
LIN {X 0,Y 601.052,Z 422.348,A -85,B 0,C 180,E1 28483.918,E2 28483.918} C_VEL
LIN {X 0,Y 601.13,Z 422.308,A -85,B 0,C 180,E1 28480.815,E2 28480.815} C_VEL
LIN {X 0,Y 601.045,Z 422.35,A -85,B 0,C 180,E1 28477.795,E2 28477.795} C_VEL
LIN {X 0,Y 601.113,Z 422.321,A -85,B 0,C 180,E1 28474.742,E2 28474.742} C_VEL
LIN {X 0,Y 601.037,Z 422.351,A -85,B 0,C 180,E1 28471.716,E2 28471.716} C_VEL
LIN {X 0,Y 601.106,Z 422.347,A -85,B 0,C 180,E1 28468.733,E2 28468.733} C_VEL
LIN {X 0,Y 601.033,Z 422.358,A -85,B 0,C 180,E1 28465.619,E2 28465.619} C_VEL
LIN {X 0,Y 601.118,Z 422.356,A -85,B 0,C 180,E1 28462.597,E2 28462.597} C_VEL
LIN {X 0,Y 601.042,Z 422.357,A -85,B 0,C 180,E1 28459.535,E2 28459.535} C_VEL
LIN {X 0,Y 601.116,Z 422.34,A -85,B 0,C 180,E1 28456.525,E2 28456.525} C_VEL
LIN {X 0,Y 601.048,Z 422.352,A -85,B 0,C 180,E1 28453.468,E2 28453.468} C_VEL
LIN {X 0,Y 601.122,Z 422.355,A -85,B 0,C 180,E1 28450.446,E2 28450.446} C_VEL
LIN {X 0,Y 601.055,Z 422.348,A -85,B 0,C 180,E1 28447.36,E2 28447.36} C_VEL
LIN {X 0,Y 601.119,Z 422.34,A -85,B 0,C 180,E1 28444.388,E2 28444.388} C_VEL
LIN {X 0,Y 601.063,Z 422.356,A -85,B 0,C 180,E1 28441.239,E2 28441.239} C_VEL
LIN {X 0,Y 601.127,Z 422.34,A -85,B 0,C 180,E1 28438.284,E2 28438.284} C_VEL
LIN {X 0,Y 601.069,Z 422.346,A -85,B 0,C 180,E1 28435.133,E2 28435.133} C_VEL
LIN {X 0,Y 601.144,Z 422.35,A -85,B 0,C 180,E1 28432.065,E2 28432.065} C_VEL
LIN {X 0,Y 601.077,Z 422.349,A -85,B 0,C 180,E1 28428.953,E2 28428.953} C_VEL
LIN {X 0,Y 601.141,Z 422.335,A -85,B 0,C 180,E1 28425.847,E2 28425.847} C_VEL
LIN {X 0,Y 601.086,Z 422.353,A -85,B 0,C 180,E1 28422.715,E2 28422.715} C_VEL
LIN {X 0,Y 601.125,Z 422.348,A -85,B 0,C 180,E1 28419.469,E2 28419.469} C_VEL
LIN {X 0,Y 601.104,Z 422.351,A -85,B 0,C 180,E1 28416.366,E2 28416.366} C_VEL
LIN {X 0,Y 601.106,Z 422.35,A -85,B 0,C 180,E1 28413.075,E2 28413.075} C_VEL
LIN {X 0,Y 601.139,Z 422.344,A -85,B 0,C 180,E1 28409.956,E2 28409.956} C_VEL
LIN {X 0,Y 601.096,Z 422.312,A -85,B 0,C 180,E1 28406.706,E2 28406.706} C_VEL
LIN {X 0,Y 601.136,Z 422.355,A -85,B 0,C 180,E1 28403.572,E2 28403.572} C_VEL
LIN {X 0,Y 601.098,Z 422.31,A -85,B 0,C 180,E1 28400.37,E2 28400.37} C_VEL
LIN {X 0,Y 601.131,Z 422.321,A -85,B 0,C 180,E1 28397.184,E2 28397.184} C_VEL
LIN {X 0,Y 601.169,Z 422.596,A -85,B 0,C 180,E1 28395.796,E2 28395.796} C_VEL
LIN {X 0,Y 609.332,Z 441.704,A -85,B 0,C 180,E1 28393.308,E2 28393.308} C_VEL
LIN {X 0,Y 615.606,Z 456.931,A -85,B 0,C 180,E1 28391.515,E2 28391.515} C_VEL
LIN {X 0,Y 626.305,Z 475.169,A -85,B 0,C 180,E1 28390.427,E2 28390.427} C_VEL
LIN {X 0,Y 628.645,Z 487.266,A -85,B 0,C 180,E1 28390.08,E2 28390.08} C_VEL
LIN {X 0,Y 623.863,Z 738.497,A -85,B 0,C 180,E1 28386.777,E2 28386.777} C_VEL
LIN {X 0,Y 621.904,Z 844.332,A -85,B 0,C 180,E1 28385.383,E2 28385.383} C_VEL
LIN {X 0,Y 620.9,Z 869.315,A -85,B 0,C 180,E1 28384.895,E2 28384.895} C_VEL
LIN {X 0,Y 619.837,Z 889.747,A -85,B 0,C 180,E1 28384.37,E2 28384.37} C_VEL
LIN {X 0,Y 618.363,Z 914.293,A -85,B 0,C 180,E1 28383.574,E2 28383.574} C_VEL
LIN {X 0,Y 616.798,Z 935.766,A -85,B 0,C 180,E1 28382.717,E2 28382.717} C_VEL
LIN {X 0,Y 615.125,Z 957.906,A -85,B 0,C 180,E1 28381.671,E2 28381.671} C_VEL
LIN {X 0,Y 613.365,Z 978.503,A -85,B 0,C 180,E1 28380.518,E2 28380.518} C_VEL
LIN {X 0,Y 611.624,Z 998.15,A -85,B 0,C 180,E1 28379.263,E2 28379.263} C_VEL
LIN {X 0,Y 609.71,Z 1018.424,A -85,B 0,C 180,E1 28377.759,E2 28377.759} C_VEL
LIN {X 0,Y 608.163,Z 1035.111,A -85,B 0,C 180,E1 28376.354,E2 28376.354} C_VEL
LIN {X 0,Y 606.354,Z 1054.357,A -85,B 0,C 180,E1 28374.502,E2 28374.502} C_VEL
LIN {X 0,Y 605.002,Z 1069.357,A -85,B 0,C 180,E1 28372.854,E2 28372.854} C_VEL
LIN {X 0,Y 603.68,Z 1084.407,A -85,B 0,C 180,E1 28370.963,E2 28370.963} C_VEL
LIN {X 0,Y 602.586,Z 1097.237,A -85,B 0,C 180,E1 28369.08,E2 28369.08} C_VEL
LIN {X 0,Y 601.671,Z 1109.688,A -85,B 0,C 180,E1 28367.007,E2 28367.007} C_VEL
LIN {X 0,Y 600.968,Z 1120.695,A -85,B 0,C 180,E1 28364.834,E2 28364.834} C_VEL
LIN {X 0,Y 600.5,Z 1129.988,A -85,B 0,C 180,E1 28362.697,E2 28362.697} C_VEL
LIN {X 0,Y 600.186,Z 1137.907,A -85,B 0,C 180,E1 28360.462,E2 28360.462} C_VEL
LIN {X 0,Y 600.03,Z 1143.491,A -85,B 0,C 180,E1 28358.529,E2 28358.529} C_VEL
LIN {X 0,Y 599.949,Z 1148.695,A -85,B 0,C 180,E1 28356.219,E2 28356.219} C_VEL
LIN {X 0,Y 599.919,Z 1152.009,A -85,B 0,C 180,E1 28354.014,E2 28354.014} C_VEL
LIN {X 0,Y 599.907,Z 1153.903,A -85,B 0,C 180,E1 28351.91,E2 28351.91} C_VEL
LIN {X 0,Y 599.885,Z 1154.394,A -85,B 0,C 180,E1 28349.522,E2 28349.522} C_VEL
LIN {X 0,Y 599.898,Z 1153.495,A -85,B 0,C 180,E1 28347.516,E2 28347.516} C_VEL
LIN {X 0,Y 599.914,Z 1151.085,A -85,B 0,C 180,E1 28345.22,E2 28345.22} C_VEL
LIN {X 0,Y 599.972,Z 1147.102,A -85,B 0,C 180,E1 28343.012,E2 28343.012} C_VEL
LIN {X 0,Y 600.048,Z 1142.219,A -85,B 0,C 180,E1 28340.988,E2 28340.988} C_VEL
LIN {X 0,Y 600.282,Z 1134.659,A -85,B 0,C 180,E1 28338.567,E2 28338.567} C_VEL
LIN {X 0,Y 600.618,Z 1127.152,A -85,B 0,C 180,E1 28336.62,E2 28336.62} C_VEL
LIN {X 0,Y 601.173,Z 1117.42,A -85,B 0,C 180,E1 28334.468,E2 28334.468} C_VEL
LIN {X 0,Y 601.949,Z 1105.684,A -85,B 0,C 180,E1 28332.303,E2 28332.303} C_VEL
LIN {X 0,Y 602.964,Z 1092.791,A -85,B 0,C 180,E1 28330.227,E2 28330.227} C_VEL
LIN {X 0,Y 604.2,Z 1078.361,A -85,B 0,C 180,E1 28328.241,E2 28328.241} C_VEL
LIN {X 0,Y 605.561,Z 1063.285,A -85,B 0,C 180,E1 28326.448,E2 28326.448} C_VEL
LIN {X 0,Y 607.149,Z 1045.865,A -85,B 0,C 180,E1 28324.647,E2 28324.647} C_VEL
LIN {X 0,Y 608.726,Z 1029.096,A -85,B 0,C 180,E1 28323.117,E2 28323.117} C_VEL
LIN {X 0,Y 610.645,Z 1008.625,A -85,B 0,C 180,E1 28321.49,E2 28321.49} C_VEL
LIN {X 0,Y 612.284,Z 990.569,A -85,B 0,C 180,E1 28320.235,E2 28320.235} C_VEL
LIN {X 0,Y 614.338,Z 967.193,A -85,B 0,C 180,E1 28318.83,E2 28318.83} C_VEL
LIN {X 0,Y 615.929,Z 947.663,A -85,B 0,C 180,E1 28317.827,E2 28317.827} C_VEL
LIN {X 0,Y 617.65,Z 924.7,A -85,B 0,C 180,E1 28316.82,E2 28316.82} C_VEL
LIN {X 0,Y 619.059,Z 902.593,A -85,B 0,C 180,E1 28316.023,E2 28316.023} C_VEL
LIN {X 0,Y 620.457,Z 878.298,A -85,B 0,C 180,E1 28315.314,E2 28315.314} C_VEL
LIN {X 0,Y 621.515,Z 855.044,A -85,B 0,C 180,E1 28314.808,E2 28314.808} C_VEL
LIN {X 0,Y 622.281,Z 830.188,A -85,B 0,C 180,E1 28314.411,E2 28314.411} C_VEL
LIN {X 0,Y 626.568,Z 591.265,A -85,B 0,C 180,E1 28311.291,E2 28311.291} C_VEL
LIN {X 0,Y 628.485,Z 485.575,A -85,B 0,C 180,E1 28309.885,E2 28309.885} C_VEL
LIN {X 0,Y 625.93,Z 474.264,A -85,B 0,C 180,E1 28309.534,E2 28309.534} C_VEL
LIN {X 0,Y 615.343,Z 456.419,A -85,B 0,C 180,E1 28308.442,E2 28308.442} C_VEL
LIN {X 0,Y 607.414,Z 437.141,A -85,B 0,C 180,E1 28306.13,E2 28306.13} C_VEL
LIN {X 0,Y 601.186,Z 422.696,A -85,B 0,C 180,E1 28304.237,E2 28304.237} C_VEL
LIN {X 0,Y 601.104,Z 422.312,A -85,B 0,C 180,E1 28303.51,E2 28303.51} C_VEL
LIN {X 0,Y 601.132,Z 422.316,A -85,B 0,C 180,E1 28300.319,E2 28300.319} C_VEL
LIN {X 0,Y 601.113,Z 422.354,A -85,B 0,C 180,E1 28297.144,E2 28297.144} C_VEL
LIN {X 0,Y 601.114,Z 422.306,A -85,B 0,C 180,E1 28293.865,E2 28293.865} C_VEL
LIN {X 0,Y 601.136,Z 422.35,A -85,B 0,C 180,E1 28290.689,E2 28290.689} C_VEL
LIN {X 0,Y 601.098,Z 422.354,A -85,B 0,C 180,E1 28287.437,E2 28287.437} C_VEL
LIN {X 0,Y 601.141,Z 422.348,A -85,B 0,C 180,E1 28284.258,E2 28284.258} C_VEL
LIN {X 0,Y 601.09,Z 422.351,A -85,B 0,C 180,E1 28281.16,E2 28281.16} C_VEL
LIN {X 0,Y 601.136,Z 422.337,A -85,B 0,C 180,E1 28278.022,E2 28278.022} C_VEL
LIN {X 0,Y 601.084,Z 422.345,A -85,B 0,C 180,E1 28274.942,E2 28274.942} C_VEL
LIN {X 0,Y 601.13,Z 422.354,A -85,B 0,C 180,E1 28271.806,E2 28271.806} C_VEL
LIN {X 0,Y 601.085,Z 422.349,A -85,B 0,C 180,E1 28268.707,E2 28268.707} C_VEL
LIN {X 0,Y 601.098,Z 422.34,A -85,B 0,C 180,E1 28265.441,E2 28265.441} C_VEL
LIN {X 0,Y 601.086,Z 422.353,A -85,B 0,C 180,E1 28262.479,E2 28262.479} C_VEL
LIN {X 0,Y 601.078,Z 422.357,A -85,B 0,C 180,E1 28259.142,E2 28259.142} C_VEL
LIN {X 0,Y 601.094,Z 422.337,A -85,B 0,C 180,E1 28256.185,E2 28256.185} C_VEL
LIN {X 0,Y 601.07,Z 422.349,A -85,B 0,C 180,E1 28253.025,E2 28253.025} C_VEL
LIN {X 0,Y 601.084,Z 422.352,A -85,B 0,C 180,E1 28250.134,E2 28250.134} C_VEL
LIN {X 0,Y 601.064,Z 422.348,A -85,B 0,C 180,E1 28246.924,E2 28246.924} C_VEL
LIN {X 0,Y 601.067,Z 422.354,A -85,B 0,C 180,E1 28244.168,E2 28244.168} C_VEL
LIN {X 0,Y 601.062,Z 422.357,A -85,B 0,C 180,E1 28240.87,E2 28240.87} C_VEL
LIN {X 0,Y 601.061,Z 422.352,A -85,B 0,C 180,E1 28238.019,E2 28238.019} C_VEL
LIN {X 0,Y 601.055,Z 422.352,A -85,B 0,C 180,E1 28234.794,E2 28234.794} C_VEL
LIN {X 0,Y 601.055,Z 422.349,A -85,B 0,C 180,E1 28231.914,E2 28231.914} C_VEL
LIN {X 0,Y 601.043,Z 422.349,A -85,B 0,C 180,E1 28228.62,E2 28228.62} C_VEL
